// TwinCAT 3 PLC project Samples
// Title: TF8040 PLC-Samples
// Company: Beckhoff Automation GmbH
// Author: Beckhoff Automation
// ProjectVersion: 2.0.0.5
// Description: PLC.Samples to demontrate function volume of TF8040.
// ProgramVersion: 3.1.4023.0
// libraries:
//   Tc2_Standard, * (Beckhoff Automation GmbH)
//   Tc2_System, * (Beckhoff Automation GmbH)
//   Tc2_Utilities, * (Beckhoff Automation GmbH)
//   Tc3_BA2, * (Beckhoff Automation GmbH)
//   Tc3_BA2_Common, * (Beckhoff Automation GmbH)
//   Tc3_BACnetRev14, * (Beckhoff Automation GmbH)
//   Tc3_Module, * (Beckhoff Automation GmbH)
// project tree:
//   / PlcTask.TcTTO
//   SAMPLES/Demo/Event/ FB_Evt_Ack.TcPOU, FB_Evt_EventClasses.TcPOU, FB_Evt_Events.TcPOU, FB_Evt_Misc.TcPOU
//   SAMPLES/Demo/Objects/ FB_Obj_AddParam.TcPOU, FB_Obj_General.TcPOU, FB_Obj_Misc.TcPOU, FB_Obj_Sequence.TcPOU, FB_Obj_UserDefined.TcPOU
//   SAMPLES/Demo/Objects/Misc/ E_UDef_Mode.TcDUT (not stored), FB_UDef_BValEx.TcPOU (not stored), FB_UDef_SpVal.TcPOU (not stored), FB_UDef_SpValEx.TcPOU (not stored)
//   SAMPLES/Demo/Optional Extensions/Events/ FB_MyLocalObjectEvents.TcPOU
//   SAMPLES/Demo/Optional Extensions/ MAIN_OPTEXT.TcPOU
//   SAMPLES/Demo/Other/ FB_Misc.TcPOU
//   SAMPLES/Demo/Plant/ FB_Plt_Init1.TcPOU, FB_Plt_Init2.TcPOU, FB_Plt_Init3.TcPOU
//   SAMPLES/Demo/Reference/ FB_Ref_Collectors.TcPOU, FB_Ref_Groups.TcPOU
//   SAMPLES/Demo/Reference/Publish and Subscribe/ FB_Ref_PubSub_Local.TcPOU, FB_Ref_PubSub_Remote.TcPOU
//   SAMPLES/Demo/Structure/ FB_Struct_Nested.TcPOU
//   SAMPLES/Demo/Supplement specific/BACnet/ FB_BACnet_RcpList.TcPOU (not stored)
//   SAMPLES/Demo/[Helper]/FunctionBlocks/Aggregates/ FB_TimerAggregateA.TcPOU, FB_ProcAggregateB.TcPOU
//   SAMPLES/Demo/[Helper]/FunctionBlocks/Nested/ FB_NestedView.TcPOU, FB_NestedView2.TcPOU, FB_SubNestedView.TcPOU, FB_SubSubNestedView.TcPOU (not stored)
//   SAMPLES/ MAIN.TcPOU
//   SAMPLES/Templates/Standard/DUTs/Enumerations/OpMod/ E_OpMod_AC.TcDUT (not stored), E_OpMod_Binary.TcDUT, E_OpMod_ClsOpn.TcDUT (not stored), E_OpMod_Step2.TcDUT (not stored)
//   SAMPLES/Templates/Standard/GVLs/ MyLabels.TcGVL, MyProfiles.TcGVL
//   SAMPLES/Templates/Standard/POUs/Trade/General/Building/ FB_BA_Bld01.TcPOU (not stored)
//   SAMPLES/Templates/Standard/POUs/Trade/General/EventClasses/ FB_BA_EC01.TcPOU
//   SAMPLES/Templates/User-defined/Objects/ FB_UDef_Obj.TcPOU (not stored)
//   SAMPLES/Templates/User-defined/Sample Weather Station/ FB_BA_MyWeatherStation.TcPOU (not stored), FB_BA_MyWeatherStationSub.TcPOU (not stored), I_BA_MyWeatherStation.TcIO (not stored), ST_BA_MyWeatherData.TcDUT (not stored)
// real-time tasks:
//   TASK PlcTask: cycle T#45ms, priority 20, ADS port 350
//   TASK Device 1 (BACnet IP)_Task_58: cycle T#40ms, priority 58, ADS port 351
//   TASK Gerät 1 (BACnet IP)_QueueTask: cycle T#2ms, priority 8, ADS port 352
// I/O:
//   DEVICE Gerät 1 (BACnet IP), AmsNetId 192.168.216.1.2.1
// variable links:
//   Samples/Samples Instance <-> Device 1 (BACnet IP)
//     PlcTask Inputs/Tc3_BACnetRev14.BACnet_Globals.DefaultAdapter.BACnet_AmsNetId <-> Inputs/AmsNetId

CONFIGURATION Samples
    RESOURCE PLC ON TwinCAT3
        TASK PlcTask(INTERVAL := T#45ms, PRIORITY := 20);
        PROGRAM MAIN WITH PlcTask : MAIN;
    END_RESOURCE
END_CONFIGURATION

// ---- SAMPLES/Templates/Standard/DUTs/Enumerations/OpMod/E_OpMod_Binary.TcDUT
{attribute 'qualified_only'}
TYPE E_OpMod_Binary :
(
	eOff			:= 0,
	eOn				:= 1
	
) UDINT;
END_TYPE

// ---- SAMPLES/Templates/Standard/GVLs/MyLabels.TcGVL
{attribute 'qualified_only'}
VAR_GLOBAL
	{region 'Functions'}
		// A
		// B
		Cmd					: FB_BA_Label			:= (sObjName:='CMD',		sDescr:='Command');
		Col					: FB_BA_Label			:= (sObjName:='KUE',		sDescr:='Kühler');
		DmprEx				: FB_BA_Label			:= (sObjName:='KL',			sDescr:='Absperrklappe Abluft');
		DmprSu				: FB_BA_Label			:= (sObjName:='KL',			sDescr:='Absperrklappe Zuluft');
		Erc					: FB_BA_Label			:= (sObjName:='WRG',		sDescr:='Wärmerückgewinnung');
		EvtCl				: FB_BA_Label			:= (sObjName:='EC',			sDescr:='Eventklasse');
		FanEx				: FB_BA_Label			:= (sObjName:='VAB',		sDescr:='Abluftventilator');
		FanSu				: FB_BA_Label			:= (sObjName:='VZU',		sDescr:='Zuluftventilator');
		// G
		// H
		// I
		// J
		// K
		// L
		// M
		// N
		// O
		PltCtrl				: FB_BA_Label			:= (sObjName:='PC',			sDescr:='Anlagensteuerung');
		PreHtr				: FB_BA_Label			:= (sObjName:='LE',			sDescr:='Lufterhitzer');
		// Q
		// R
		// S	
		Trnd				: FB_BA_Label			:= (sObjName:='TR',			sDescr:='Trend');
		// U
		// v
		// W
		// X
		// Y
		// Z
	{endregion}
	{region 'Aggregates'}
		// A
		// B
		// C
		// D
		// E
		// F
		// G
		// H
		// I
		// J
		// K
		// L
		// M
		// N
		// O
		// P	
		// Q
		// R
		// S	
		// t
		// U
		// v
		// W
		// X
		// Y
		// Z
	{endregion}
	{region 'Processes'}
		ProcPreRinse		: FB_BA_LabelProcess	:= (sProcessName:='Vorspülen');
		ProcDriveDamper		: FB_BA_LabelProcess	:= (sProcessName:='Klappen fahren');
	{endregion}
END_VAR

// ---- SAMPLES/Templates/Standard/GVLs/MyProfiles.TcGVL
{attribute 'qualified_only'}
VAR_GLOBAL
	{region 'Placeholder'}
		{region 'Text'}
			txtOff						: STRING						:= 'Aus';
			txtOn						: STRING						:= 'Ein';
			txtNormal					: STRING						:= 'Normal';
			txtOffnormal				: STRING						:= 'Unnormal';
			txtAlert					: STRING						:= 'Alarm';
			txtDisturb					: STRING						:= 'Störung';
			txtExceeded					: STRING						:= 'Überschritten';
			txtMonitoring				: STRING						:= 'Überwachung';
			txtProtection				: STRING						:= 'Schutzbetrieb';
			txtEconomy					: STRING						:= 'Economy';
			txtComfort					: STRING						:= 'Comfort';
		{endregion}
		{region 'Event Transition Text'}
			trnsExceeded				: T_BA_EventTransitionText		:= [txtExceeded,			txtDisturb,			txtNormal];
			trnsMonitoring				: T_BA_EventTransitionText		:= [txtMonitoring,			txtDisturb,			txtNormal];
		{endregion}
		{region 'Multistate Text'}
			txtEnergyLevel				: T_BA_StateTextArray			:= [txtProtection,			txtEconomy,			txtComfort];
		{endregion}
	{endregion}
END_VAR
VAR_GLOBAL
	{region 'Sample Templates'}
		// A
		// B
		CmdB							: FB_BA_ProfileBEvtObj			:= (sInactiveText := txtOff,			sActiveText := txtOn,			aEventTransitionText := trnsMonitoring,							nEventClassID := 11);
		// D
		// E
		// F
		// G
		// H
		// I
		// J
		// K
		// L
		// M
		// N
		// O
		// P	
		// Q
		// R
		// S	
		// t
		// U
		// v
		// W
		// X
		// Y
		// Z
	{endregion}
	{region 'Sample Objects'}
		{region 'Analog'}
			AV_Prf						: FB_BA_ProfileAEvtObj			:= (eUnit:=E_BA_Unit.eTemperature_DegreesCelsius,						aEventTransitionText:=MyProfiles.trnsExceeded,					nEventClassID:=11);
			AVOp_Prf					: FB_BA_ProfileAObj				:= (eUnit:=E_BA_Unit.eTemperature_DegreesCelsius);
			AI_Prf						: FB_BA_ProfileAEvtObj			:= (eUnit:=E_BA_Unit.eTemperature_DegreesCelsius,						aEventTransitionText:=MyProfiles.trnsExceeded,					nEventClassID:=11);
			AO_Prf						: FB_BA_ProfileAEvtObj			:= (eUnit:=E_BA_Unit.eTemperature_DegreesCelsius,						aEventTransitionText:=MyProfiles.trnsExceeded,					nEventClassID:=11);
		{endregion}
		{region 'Binary'}
			BV_Prf						: FB_BA_ProfileBEvtObj			:= (sInactiveText := txtOff, sActiveText := txtOn,						aEventTransitionText:=MyProfiles.trnsExceeded,					nEventClassID:=11);
			BVOp_Prf					: FB_BA_ProfileBObj				:= (sInactiveText := txtOff, sActiveText := txtOn);
			BI_Prf						: FB_BA_ProfileBEvtObj			:= (sInactiveText := txtOff, sActiveText := txtOn,						aEventTransitionText:=MyProfiles.trnsExceeded,					nEventClassID:=11);
			BO_Prf						: FB_BA_ProfileBEvtObj			:= (sInactiveText := txtOff, sActiveText := txtOn,						aEventTransitionText:=MyProfiles.trnsExceeded,					nEventClassID:=11);
		{endregion}
		{region 'Multistate'}
			MV_Prf						: FB_BA_ProfileMEvtObj			:= (aStateText:=MyProfiles.txtEnergyLevel,								aEventTransitionText:=MyProfiles.trnsExceeded,					nEventClassID:=11);	
			MVOp_Prf					: FB_BA_ProfileMObj				:= (aStateText:=MyProfiles.txtEnergyLevel);
			MI_Prf						: FB_BA_ProfileMEvtObj			:= (aStateText:=MyProfiles.txtEnergyLevel,								aEventTransitionText:=MyProfiles.trnsExceeded,					nEventClassID:=11);
			MO_Prf						: FB_BA_ProfileMEvtObj			:= (aStateText:=MyProfiles.txtEnergyLevel,								aEventTransitionText:=MyProfiles.trnsExceeded,					nEventClassID:=11);
		{endregion}
		{region 'Misc'}
			Loop_Prf					: FB_BA_ProfileAObj				:= (eUnit:=E_BA_Unit.eOther_Percent);
			Cal_Prf						: FB_BA_ProfileBObj				:= (sInactiveText := txtOff, sActiveText := txtOn);
			SchedA_Prf					: FB_BA_ProfileAObj				:= (eUnit:=E_BA_Unit.eOther_Percent);
			SchedB_Prf					: FB_BA_ProfileBObj				:= (sInactiveText := txtOff, sActiveText := txtOn);
			SchedM_Prf					: FB_BA_ProfileMObj				:= (aStateText:=MyProfiles.txtEnergyLevel);
			Trend_Prf					: FB_BA_ProfileBObj				:= (sInactiveText := txtOff, sActiveText := txtOn);
			EvtCls_Prf					: FB_BA_Profile;
		{endregion}
		{region 'Custom'}
			MyWthSt_Prf					: FB_BA_Profile;
		{endregion}
		{region 'Collectors'}
			Col_PrfEn					: FB_BA_ProfileBObj				:= (sInactiveText := 'Nein', sActiveText := 'Ja');
			Col_PrfValA					: FB_BA_ProfileAObj				:= (eUnit:=E_BA_Unit.eTemperature_DegreesCelsius);
		{endregion}
	{endregion}
END_VAR

// ---- SAMPLES/MAIN.TcPOU
PROGRAM MAIN
VAR
	{region 'Settings'}
		DPAD					: FB_BA_CarelessDPAD:=(
									aIdentifier:=[
										(* Level 1 *)	(eNodeType:=E_BA_NodeType.eBuilding,	nIndexDigits:=2),
										(* Level 2 *)	(eNodeType:=E_BA_NodeType.eTrade,		nIndexDigits:=0),
										(* Level 3 *)	(eNodeType:=E_BA_NodeType.ePlant,		nIndexDigits:=2,			sSeparator_ObjectName:='~~~',		sSeparator_Description:=' --- '),
										(* Level 4 *)	(eNodeType:=E_BA_NodeType.eAggregate,	nIndexDigits:=2,			sSeparator_ObjectName:='++'),
										(* Level 5 *)	(eNodeType:=E_BA_NodeType.eFunction,	nIndexDigits:=3)
								]);
	{endregion}
		 
	Smpl						: FB_BA_View			:= (									sDescription:='Samples');
	{region 'Demonstration'}
		Demo					: FB_BA_View			:= (iParent:=Smpl,						sDescription:='Demonstration');
			Obj					: FB_BA_View			:= (iParent:=Demo,						sDescription:='Objects');
				General			: FB_Obj_General		:= (iParent:=Obj,						sDescription:='General objects');
				Misc			: FB_Obj_Misc			:= (iParent:=Obj,						sDescription:='Miscellaneous objects');
				Seq				: FB_Obj_Sequence		:= (iParent:=Obj,						sDescription:='Sequences');
				UdObj			: FB_Obj_UserDefined	:= (iParent:=Obj,						sDescription:='User defined objects');
				AddParam		: FB_Obj_AddParam		:= (iParent:=Obj,						sDescription:='Additional parameters');
					 
			Ref					: FB_BA_View			:= (iParent:=Demo,						sDescription:='Reference');
				Collect			: FB_Ref_Collectors		:= (iParent:=Ref,						sDescription:='Collectors');
				Groups			: FB_Ref_Groups			:= (iParent:=Ref,						sDescription:='Groups');
				PubSubLc		: FB_Ref_PubSub_Local	:= (iParent:=Ref,						sDescription:='Publisher and subscriber (Local)');
				PubSubRm		: FB_Ref_PubSub_Remote	:= (iParent:=Ref,						sDescription:='Publisher and subscriber (Remote)');
					 
			Evt					: FB_BA_View			:= (iParent:=Demo,						sDescription:='Event');
				EvtCls			: FB_Evt_EventClasses	:= (iParent:=Evt,						sDescription:='Event classes');
				Events			: FB_Evt_Events			:= (iParent:=Evt,						sDescription:='Events');
				Ack				: FB_Evt_Ack			:= (iParent:=Evt,						sDescription:='Acknowledgement');
				MiscEvt			: FB_Evt_Misc			:= (iParent:=Evt,						sDescription:='Miscellaneous');
					 
			Strct				: FB_BA_View			:= (iParent:=Demo,						sDescription:='Structure');
				Nested			: FB_Struct_Nested		:= (iParent:=Strct,						sDescription:='Nested objects');
					 
			Plt					: FB_BA_View			:= (iParent:=Demo,						sDescription:='Plant');
				PltCtrl1		: FB_Plt_Init1			:= (iParent:=Plt,						sDescription:='Plant control initialization 1');
				PltCtrl2		: FB_Plt_Init2			:= (iParent:=Plt,						sDescription:='Plant control initialization 2');
				PltCtrl3		: FB_Plt_Init3			:= (iParent:=Plt,						sDescription:='Plant control initialization 3');
					 
			Spl					: FB_BA_View			:= (iParent:=Demo,						sDescription:='Supplement specific');
				BACnet_RcpList	: FB_BACnet_RcpList		:= (iParent:=Spl,						sDescription:='Recipient list (BACnet)');
					 
			Other				: FB_BA_View			:= (iParent:=Demo,						sDescription:='Other');
				MscOth			: FB_Misc				:= (iParent:=Other,						sDescription:='Miscellaneous');
	{endregion}
	{region 'Templates'}
		Tmpl					: FB_BA_View			:= (iParent:=Smpl,						sDescription:='Templates');
			Gen					: FB_BA_View			:= (iParent:=Tmpl,						sDescription:='General');
				Bld01			: FB_BA_Bld01			:= (iParent:=Gen,						sDescription:='Building information');
				EvtCls01		: FB_BA_EC01			:= (iParent:=Gen,						sDescription:='Event Classes');
	{endregion}		
END_VAR
VAR		
	nCounter					: UDINT					:= 0;	
END_VAR

nCounter:=(nCounter+1);

Smpl();

// Demonstration:
Demo();

Obj();
General();
Misc();
Seq();
UdObj();
AddParam();

Ref();
Collect();
Groups();
PubSubLc();
PubSubRm();

Evt();
EvtCls();
Events();
Ack();
MiscEvt();

Strct();
Nested();

Plt();
PltCtrl1();
PltCtrl2();
PltCtrl3();

Spl();
BACnet_RcpList();

Other();
MscOth();

// Templates:
Tmpl();

Gen();
Bld01();
EvtCls01();

// Optional extensions:
MAIN_OPTEXT();

END_PROGRAM

// ---- SAMPLES/Demo/Objects/FB_Obj_General.TcPOU
// Demonstration of objects.
// > See "FB_BA_EC01" to view decleared event classes.
FUNCTION_BLOCK FB_Obj_General EXTENDS FB_BA_View
VAR
	{region 'Analog'}
		A										: FB_BA_View := (
													iParent									:= THIS^,
													sDescription							:= '{Analog objects}'
												);
			 
			// Intention:						Value
			AV									: FB_BA_AV := (
													iParent									:= A,
													sDescription							:= '{Analog Value}',
													eUnit									:= E_BA_Unit.eOther_Percent,
													nEventClassID							:= 11,
													stLowLimit								:= F_BA_Limit(TRUE, 0),
													stHighLimit								:= F_BA_Limit(TRUE, 50),
													stTimeDelay								:= F_BA_TimeDelay(1, 1),
													bEnPgm									:= TRUE,
													fValPgm									:= 10.0
												);
													
			// Intention:						Value for Display
			// Operation:						Display
			fAVDsp_ValuePgm						: REAL := 0;
			AVDsp								: FB_BA_AV_Op := (
													iParent									:= A,
													sObjectName								:= '{MyAvDsp}',
													sDescription							:= '{Sample AV Display}',
													eUnit									:= E_BA_Unit.eOther_Percent
												);	
			
			// Intention:						Value for Setpoint
			// Operation:						Setpoint
			AVSp								: FB_BA_AV_Op := (
													iParent									:= A,
													sDescription							:= '{Sample AV Setpoint}',
													eUnit									:= E_BA_Unit.eTemperature_DegreesCelsius,
													fValueRm								:= 3
												);
			bAVSp2_ValViaProp					: BOOL;
			fAVSp2_ValViaProp					: REAL;
			AVSp2								: FB_BA_AV_Op := (
													iParent									:= A,
													sDescription							:= '{Sample AV Setpoint 2}',
													eUnit									:= E_BA_Unit.eTemperature_DegreesCelsius,
													fValueRm								:= 3
												);
		
			// Intention:						Input
			// Hardware:						Process Data
			fAI_Proc_ValuePgm					: REAL := 20;
			AI_Proc								: FB_BA_AI := (
													iParent									:= A,
													sDescription							:= '{Sample AI (Process Data)}',
													sDeviceType								:= 'Analoger Eingang',
													eUnit									:= E_BA_Unit.eOther_Percent,
													nEventClassID							:= 11
												);
		
			// Intention:						Input
			// Hardware:						Raw Data
			AI_Raw								: FB_BA_AI_Raw := (
													iParent									:= A,
													sDescription							:= '{Sample AI (Raw)}',
													sDeviceType								:= 'Analoger Eingang',
													eUnit									:= E_BA_Unit.eOther_Percent,
													nEventClassID							:= 11
												);
		
			// Intention:						Input
			// Hardware:						I/O
			AI_IO								: FB_BA_AI_IO := (
													iParent									:= A,
													sDescription							:= '{Sample AI (IO)}',
													sDeviceType								:= 'Analoger Eingang',
													eUnit									:= E_BA_Unit.eOther_Percent,
													nEventClassID							:= 11
												);
												
			AI_IO_2_10V							: FB_BA_AI_IO := (
													iParent									:= A,
													sDescription							:= '{Sample AI (IO)}',
													sDeviceType								:= 'Analoger Eingang (2-10V)',
													eUnit									:= E_BA_Unit.eOther_Percent,
													nEventClassID							:= 11
												);
		
			// Intention:						Input
			// Hardware:						I/O
			AI_Temp								: FB_BA_AI_IOEx := (
													iParent									:= A,
													sDescription							:= '{Sample AI Temperaturfühler (Temp)}',
													sDeviceType								:= 'Temperaturfühler',
													eUnit									:= E_BA_Unit.eTemperature_DegreesCelsius,
													eSensor									:= E_BA_MeasuringElement.eNI1000,
													nEventClassID							:= 11
												);
		
			// Intention:						Input for Display
			// Operation:						Display
			// Hardware:						I/O
			// Parameter:						EventDetectionEnable = FALSE
			AIDsp_IO							: FB_BA_AI_IO := (
													iParent									:= A,
													sDescription							:= '{Sample AI Display (IO)}',
													sDeviceType								:= 'Analoger Eingang',
													eUnit									:= E_BA_Unit.eOther_Percent,
													bEventDetectionEnable					:= FALSE,
													nEventClassID							:= 11
												);
		
			// Intention:						Output
			// Hardware:						Process Data
			AO_CmdProc							: FB_BA_AO := (
													iParent									:= A,
													sDescription							:= '{Analog Befehl (Process Data)}',
													eUnit									:= E_BA_Unit.eOther_Percent,
													nEventClassID							:= 11
												);
		
			// Intention:						Output
			// Hardware:						Raw Data
			AO_CmdRaw							: FB_BA_AO_Raw := (
													iParent									:= A,
													sDescription							:= '{Analog Befehl (Raw Data)}',
													eUnit									:= E_BA_Unit.eOther_Percent,
													nEventClassID							:= 11
												);
		
			// Intention:						Output
			// Hardware:						I/O
			AO_CmdIO							: FB_BA_AO_IO := (
													iParent									:= A,
													sDescription							:= '{Analog Befehl (IO)}',
													eUnit									:= E_BA_Unit.eOther_Percent,
													nEventClassID							:= 11
												);
		
			// Intention:						Output for Display
			// Operation:						Display
			// Hardware:						I/O
			// Parameter:						EventDetectionEnable = FALSE
			AODisp_CmdIO						: FB_BA_AO_IO := (
													iParent									:= A,
													sDescription							:= '{Analog Befehl Display (IO)}',
													eUnit									:= E_BA_Unit.eOther_Percent,
													bEventDetectionEnable					:= FALSE,
													nEventClassID							:= 11
												);
	{endregion}
	{region 'Binary'}
		B										: FB_BA_View := (
													iParent									:= THIS^,
													sDescription							:= '{Binary objects}'
												);
			 
			// Intention:						Value
			BV									: FB_BA_BV := (
													iParent									:= B,
													sDescription							:= '{Binary Value}',
													sInactiveText							:= 'Aus',
													sActiveText								:= 'Ein',
													nEventClassID							:= 10
												);
															
			// Intention:						Value for Display
			// Operation:						Display
			bBVDsp_ValuePgm						: BOOL := FALSE;
			BVDsp								: FB_BA_BV_Op := (
													iParent									:= B,
													sDescription							:= '{Sample BV Display}',
													sInactiveText							:= 'Aus',
													sActiveText								:= 'Ein'
												);
			
			// Intention:						Value for Setpoint
			// Operation:						Setpoint
			BVSp								: FB_BA_BV_Op := (
													iParent									:= B,
													sDescription							:= '{Sample BV Setpoint}',
													sInactiveText							:= 'Aus',
													sActiveText								:= 'Ein',
													bValueRm								:= TRUE
												);
												
			// Intention:						Value for Setpoint
			// Operation:						Pushbutton
			nBVPushButton_Counter				: UINT;
			BVPushButton						: FB_BA_BV_Op := (
													iParent									:= B,
													sDescription							:= '{Sample BV Pushbutton}',
													sInactiveText							:= 'Aus',
													sActiveText								:= 'Ein',
													eToggleMode								:= E_BA_ToggleMode.ePushButton
												);
		
			// Intention:						Input
			// Hardware:						Process Data
			BI_Proc								: FB_BA_BI := (
													iParent									:= B,
													sDescription							:= '{Sample BI (Process Data)}',
													sDeviceType								:= 'Sicherung',
													sInactiveText							:= 'Normal',
													sActiveText								:= 'Ausgelöst',
													nEventClassID							:= 11
												);
		
			// Intention:						Input
			// Hardware:						Raw Data
			BI_Raw								: FB_BA_BI_Raw := (
													iParent									:= B,
													sDescription							:= '{Sample BI (Raw Data)}',
													sDeviceType								:= 'Sicherung',
													sInactiveText							:= 'Normal',
													sActiveText								:= 'Ausgelöst',
													nEventClassID							:= 11
												);
		
			// Intention:						Input
			// Hardware:						I/O
			BI_DstbIO							: FB_BA_BI_IO := (
													iParent									:= B,
													sDescription							:= '{Sample BI Disturb (IO)}',
													sDeviceType								:= 'Sicherung',
													sInactiveText							:= 'Normal',
													sActiveText								:= 'Ausgelöst',
													ePolarity								:= E_BA_Polarity.eReverse,
													nEventClassID							:= 51,
													eEnPlantLock							:= E_BA_LockPriority.eLocalMedium
												);
		
			// Intention:						Input for Display
			// Operation:						Display
			// Hardware:						I/O
			// Parameter:						EventDetectionEnable = FALSE
			BIDsp_SwiIO							: FB_BA_BI_IO := (
													iParent									:= B,
													sDescription							:= '{Sample BI Schalter Display (IO)}',
													sDeviceType								:= 'Sicherung',
													sInactiveText							:= 'Normal',
													sActiveText								:= 'Ausgelöst',
													ePolarity								:= E_BA_Polarity.eReverse,
													nEventClassID							:= 182,
													bEventDetectionEnable					:= FALSE
												);
		
			// Intention:						Output
			// Hardware:						I/O
			BO_CmdIO							: FB_BA_BO_IO := (
													iParent									:= B,
													sDescription							:= '{Sample BO Befehl (IO)}',
													sInactiveText							:= 'Aus',
													sActiveText								:= 'Ein',
													nEventClassID							:= 11,
													stTimeDelay := (
														nToAbnormal							:= 3
													)
												);
		
			// Intention:						Output
			// Hardware:						Process Data
			BO_CmdProc							: FB_BA_BO := (
													iParent									:= B,
													sDescription							:= '{Sample BO Befehl (Process Data)}',
													sInactiveText							:= 'Aus',
													sActiveText								:= 'Ein',
													nEventClassID							:= 11,
													stTimeDelay := (
														nToAbnormal							:= 3
													)
												);
		
			// Intention:						Output
			// Hardware:						Raw Data
			BO_CmdRaw							: FB_BA_BO_Raw := (
													iParent									:= B,
													sDescription							:= '{Sample BO Befehl (Raw Data)}',
													sInactiveText							:= 'Aus',
													sActiveText								:= 'Ein',
													nEventClassID							:= 11,
													stTimeDelay := (
														nToAbnormal							:= 3
													)
												);
													
			// Intention:						Output for Display
			// Operation:						Display
			// Hardware:						I/O
			// Parameter:						EventDetectionEnable = FALSE
			BODisp_CmdIO						: FB_BA_BO_IO := (
													iParent									:= B,
													sDescription							:= '{Sample BO Befehl Display (IO)}',
													sInactiveText							:= 'Aus',
													sActiveText								:= 'Ein',
													nEventClassID							:= 182,
													bEventDetectionEnable					:= FALSE
												);
	{endregion}
	{region 'Multistate'}
		M										: FB_BA_View := (
													iParent									:= THIS^,
													sDescription							:= '{Multistate objects}'
												);
			 
			// Intention:						Value
			MV									: FB_BA_MV := (
													iParent									:= M,
													sDescription							:= '{Sample MV}',
													aStateText								:= [ 'Aus', 'Stufe 1', 'Stufe 2' ],
													nEventClassID							:= 11
												);
			
			// Intention:						Value for Display
			// Operation:						Display
			nAVDsp_ValuePgm						: UDINT := 1;
			MVDsp								: FB_BA_MV_Op := (
													iParent									:= M,
													sObjectName								:= '{BAS01}',
													sDescription							:= '{Sample MV Display}',
													aStateText								:= [ 'Auto', 'Aus', 'Stufe 1', 'Stufe 2' ]
												);
			
			// Intention:						Value for Setpoint
			// Operation:						Setpoint
			MVSp								: FB_BA_MV_Op := (
													iParent									:= M,
													sObjectName								:= '{BAM01}',
													sDescription							:= '{Sample MV Setpoint}',
													aStateText								:= [ 'Auto', 'Aus', 'Stufe 1', 'Stufe 2' ],
													nValueRm								:= 1
												);
												
												
			nMVPushButton_Counter				: UDINT;
			MVPushButton						: FB_BA_MV_Op := (
													iParent									:= M,
													sDescription							:= '{Sample MV Pushbutton}',
													aStateText								:= [ 'Aus', 'Increment 1', 'Increment 2' ],
													eToggleMode								:= E_BA_ToggleMode.ePushButton
												);
		
			// Intention:						Input
			// Hardware:						Process Data
			MI_StateProc						: FB_BA_MI := (
													iParent									:= M,
													sDescription							:= '{Sample MI State (Process Data)}',
													sDeviceType								:= 'Gerät',
													aStateText								:= [ 'Aus', 'Stufe 1', 'Stufe 2', 'Stufe 3', 'Stufe 4' ],
													aAlarmValues							:= [ 3, 4 ],
													aFaultValues							:= [ 5 ],
													nEventClassID							:= 11
												);
		
			// Intention:						Input
			// Hardware:						Raw Data
			MI_StateRaw							: FB_BA_MI_Raw := (
													iParent									:= M,
													sDescription							:= '{Sample MI State (Raw Data)}',
													sDeviceType								:= 'Gerät',
													aStateText								:= [ 'Aus', 'Stufe 1', 'Stufe 2', 'Stufe 3', 'Stufe 4' ],
													aAlarmValues							:= [ 3, 4 ],
													aFaultValues							:= [ 5 ],
													nEventClassID							:= 11
												);
		
			// Intention:						Input
			// Hardware:						I/O
			MI_StateIO							: FB_BA_MI_IO := (
													iParent									:= M,
													sDescription							:= '{Sample MI State (IO)}',
													sDeviceType								:= 'Gerät',
													aStateText								:= [ 'Aus', 'Stufe 1', 'Stufe 2', 'Stufe 3', 'Stufe 4' ],
													aAlarmValues							:= [ 3, 4 ],
													aFaultValues							:= [ 5 ],
													nEventClassID							:= 11
												);
		
			// Intention:						Input for Display
			// Operation:						Display
			// Hardware:						I/O
			// Parameter:						EventDetectionEnable = FALSE
			MIDsp_Swi_StateIO					: FB_BA_MI_IO := (
													iParent									:= M,
													sDescription							:= '{Sample MI State (IO)}',
													sDeviceType								:= 'Gerät',
													aStateText								:= [ 'Zustand 1', 'Zustand 2', 'Zustand 3', 'Unbekannt' ],
													nEventClassID							:= 182,
													bEventDetectionEnable					:= FALSE
												);
		
			// Intention:						Output for Display
			// Operation:						Display
			// Hardware:						I/O
			// Parameter:						EventDetectionEnable = FALSE
			MODisp_IO							: FB_BA_MO_IO := (
													iParent									:= M,
													sDescription							:= '{Sample MO Befehl (IO)}',
													aStateText								:= [ 'Aus', 'Stufe 1', 'Stufe 2', 'Stufe 3', 'Stufe 4' ],
													nEventClassID							:= 182,
													bEventDetectionEnable					:= FALSE
												);
		
			// Intention:						Output
			// Hardware:						Process Data
			MO_CmdProc							: FB_BA_MO := (
													iParent									:= M,
													sDescription							:= '{Sample MO Befehl (Process Data)}',
													aStateText								:= [ 'Aus', 'Stufe 1', 'Stufe 2', 'Stufe 3', 'Stufe 4' ],
													nEventClassID							:= 182
												);
		
			// Intention:						Output
			// Hardware:						Raw Data
			MO_CmdRaw							: FB_BA_MO_Raw := (
													iParent									:= M,
													sDescription							:= '{Sample MO Befehl (Raw Data)}',
													aStateText								:= [ 'Aus', 'Stufe 1', 'Stufe 2', 'Stufe 3', 'Stufe 4' ],
													nEventClassID							:= 182
												);
	{endregion}
END_VAR

SUPER^();

// Analog:
A();

AV();
AVDsp(fValuePgm	:= MAX(fAVDsp_ValuePgm, AVSp.fPresentValue));
AVSp();
IF (bAVSp2_ValViaProp) THEN
	bAVSp2_ValViaProp := FALSE;
	AVSp2.PresentValue := fAVSp2_ValViaProp;
END_IF
AVSp2();
AI_Proc(fVal := fAI_Proc_ValuePgm);
AI_Raw();
AI_IO();
AI_IO_2_10V();
AI_Temp();
AIDsp_IO();
AO_CmdProc();
AO_CmdRaw();
AO_CmdIO();
AODisp_CmdIO();

// Binary:
B();

BV(bEnCrit := BI_DstbIO.bEvent);
BVDsp(bValuePgm	:= (bBVDsp_ValuePgm OR BVSp.bPresentValue));
BVSp();
BVPushButton();
BI_Proc();
BI_Raw();
BI_DstbIO();
BIDsp_SwiIO();
BO_CmdProc();
BO_CmdRaw();
BO_CmdIO();
BODisp_CmdIO();

IF (BVPushButton.bPresentValue <> BVPushButton.bDefaultValue) THEN
	nBVPushButton_Counter := (nBVPushButton_Counter+1);
END_IF

// Multistate:
M();

MV();
MVDsp(nValuePgm := MAX(nAVDsp_ValuePgm, MVSp.nPresentValue));
MVSp();
MVPushButton();
MI_StateProc();
MI_StateRaw();
MI_StateIO();
MIDsp_Swi_StateIO();
MODisp_IO(
	bEnPgm		:= TRUE,
	nValPgm		:= LIMIT(1, TO_UDINT(AVSp.fPresentValue), MODisp_IO.StateCount)
);
MO_CmdProc();
MO_CmdRaw();

IF (MVPushButton.nPresentValue <> MVPushButton.nDefaultValue) THEN
	nMVPushButton_Counter := (nMVPushButton_Counter+(MVPushButton.nPresentValue-1));
END_IF

END_FUNCTION_BLOCK

// ---- SAMPLES/Demo/Objects/FB_Obj_Misc.TcPOU
// Demonstration of objects.
// > See "FB_BA_EC01" to view decleared event classes.
FUNCTION_BLOCK FB_Obj_Misc EXTENDS FB_BA_View
VAR CONSTANT
	TREND_COUNT									: INT										:= 10;
END_VAR
VAR
	{region 'Project'}
		Proj									: FB_BA_View := (
													iParent									:= THIS^,
													sDescription							:= '{Project information}'
												);
				 
			// Intention:						Project Information
			Project								: FB_BA_Project := (
													iParent									:= Proj,
													sDescription							:= '{My project infos}',
													stProject := (	
														sTitle								:= 'Mein Projekt',
														sDescription						:= 'PLC Beispielprojekt',
														sLocation							:= 'Verl'
													)
												);
	{endregion}
	{region 'Loop'}
		Loop									: FB_BA_View := (
													iParent									:= THIS^,
													sDescription							:= '{Loop objects}'
												);
				 
			fLoop_Setpoint						: REAL										:= 20;								// Temperature setpoint.
			fLoop_CtrlVal						: REAL										:= 16;								// Simulation of controlled variable value.

			// Initialization:					Single loop for heating.
			Heat_En								: REFERENCE TO BOOL							REF= Heat.bEn;
			Heat_EnSync							: REFERENCE TO BOOL							REF= Heat.bEnSync;
			Heat_ValSync						: REFERENCE TO REAL							REF= Heat.fValSync;
			Heat_Y								: REFERENCE TO REAL							REF= Heat.fPresentValue;
			Heat								: FB_BA_Loop := (
													iParent									:= Loop,
													sDescription							:= '{Heating Loop}',
													eOutputUnit								:= E_BA_Unit.eOther_Percent,
													bEn										:= TRUE,
													eActionRm								:= E_BA_Action.eReverse,
													fProportionalConstant					:= 3.0,
													fIntegralConstant						:= 180
												);

			// Initialization:					Single loop for heating.
			Cool_En								: REFERENCE TO BOOL							REF= Cool.bEn;
			Cool_EnSync							: REFERENCE TO BOOL							REF= Cool.bEnSync;
			Cool_ValSync						: REFERENCE TO REAL							REF= Cool.fValSync;
			Cool_Y								: REFERENCE TO REAL							REF= Cool.fPresentValue;
			Cool								: FB_BA_Loop := (
													iParent									:= Loop,
													sDescription							:= '{Cooling Loop}',
													eOutputUnit								:= E_BA_Unit.eOther_Percent,
													bEn										:= TRUE,
													eActionRm								:= E_BA_Action.eDirect,
													fProportionalConstant					:= 3.0,
													fIntegralConstant						:= 180
												);
	{endregion}
	{region 'Calendar'}
		Cals									: FB_BA_View := (
													iParent									:= THIS^,
													sDescription							:= '{Calendar objects}'
												);

			// Intention:						Initialize calendar parameters with parameter builders.
			// Parameter:						tWeek										= F_BA_CalendarBuilder()
			Cal1								: FB_BA_Cal := (
													iParent									:= Cals,
													sDescription							:= '{Calendar 1}',
													aDateList								:= F_BA_CalendarBuilder()
																								.AppendDate(2021, E_BA_Month.eMarch, 10)
																								.AppendDateRange(nFromYear := 2021,E_BA_Month.eMarch,10, nToYear := 2021,E_BA_Month.eMarch,15)
																								.AppendWeekNDay(E_BA_Weekday.eMonday, E_BA_Week.Unspecified, E_BA_Month.Unspecified)
																								.Build()
												);
													 
			// Intention:						Initialize calendar parameters with helper methods.
			//									aDateList									= [(..., F_BA_DateVal(...)), (..., F_BA_DateRangeVal(...)), (..., F_BA_WeekNDayVal(...))]
			Cal2								: FB_BA_Cal := (
													iParent									:= Cals,
													sDescription							:= '{Calendar 2}',
													aDateList := [(
														eType								:= E_BA_DateValChoice.eDate,
														uDate								:= F_BA_DateVal(2020,E_BA_Month.eDecember,10)
													),(
														eType								:= E_BA_DateValChoice.eDateRange,
														uDate								:= F_BA_DateRangeVal(nFromYear:=2020,E_BA_Month.eMarch,5, nToYear:=2020,E_BA_Month.eMarch,10)
													),(
														eType								:= E_BA_DateValChoice.eWeekNDay,
														uDate								:= F_BA_WeekNDayVal(E_BA_Weekday.eTuesday, E_BA_Week.Unspecified, E_BA_Month.Unspecified)
													)]
												);

			Cal3								: FB_BA_Cal := (
													iParent									:= Cals,
													sDescription							:= '{Calendar 3}'
												);
	{endregion}
	{region 'Scheduler'}
		Sched									: FB_BA_View := (
													iParent									:= THIS^,
													sDescription							:= '{Schedule objects}'
												);
			
			// Intention:						Initialize scheduler parameters with parameter builders.
			// Parameter:						tWeek										= F_BA_WeeklyScheduleBuilder()
			//									tCalendar									= F_BA_ScheduleCalendarBuilder()
			//									tException									= F_BA_ExceptionScheduleBuilder()
			SchedA								: FB_BA_SchedA := (
													iParent									:= Sched,
													sDescription							:= '{Schedule Analog}',
													eUnit									:= E_BA_Unit.eTemperature_DegreesCelsius,
													aWeek									:= F_BA_WeeklyScheduleBuilder()
																								.SetAllDays()
																									.AppendA(T#0H, 1.0)
																									.Close()
																								.SetDay(E_BA_Weekday.eMonday)
																									.AppendA(T#0H, 2.0).AppendA(T#8H, 3.0).AppendA(T#16H, 2.0)
																									.Close()
																								.SetDayRange(E_BA_Weekday.eSaturday, E_BA_Weekday.eSunday)
																									.AppendA(T#0H, 4.0)
																									.Close()
																								.Build(),
													aCalendar								:= F_BA_ScheduleCalendarBuilder()
																								.AppendReference(Cal1)
																									.AppendA(T#0H, 1.0).AppendA(T#6H, 2.0).AppendNull(T#12H)
																									.Close()
																								.AppendReference(Cal2)
																									.AppendA(T#10H, 1.0).AppendNull(T#12H)
																									.Close()
																								.Build(),
													aException								:= F_BA_ExceptionScheduleBuilder()
																								.AppendDate(2021, E_BA_Month.eMarch, 10)
																									.AppendA(T#0H, 1.0).AppendA(T#6H, 2.0).AppendNull(T#12H)
																									.Close()
																								.AppendDateRange(nFromYear := 2021,E_BA_Month.eMarch,10, nToYear := 2021,E_BA_Month.eMarch,15)
																									.AppendA(T#12H, 1.0).AppendNull(T#16H)
																									.Close()
																								.AppendWeekNDay(E_BA_Weekday.eFriday, E_BA_Week.Unspecified, E_BA_Month.Unspecified)
																									.AppendA(T#20H, 3.0)
																									.Close()
																								.Build()
												);
			
			// Intention:						Initialize scheduler parameters with helper methods.
			// Parameter:						tWeek										= F_BA_SchedWeeklyXxA(...)
			//									tCalendar									= F_BA_SchedCalendar(...)
			//									tException									= [(..., F_BA_SchedEntryXxA(...)), (..., F_BA_SchedEntryXxA(...)), (..., F_BA_SchedEntryXxA(...))]
			SchedB								: FB_BA_SchedB := (
													iParent									:= Sched,
													sDescription							:= '{Schedule Bool}',
													sInactiveText							:= 'Aus',
													sActiveText								:= 'Ein',
													aWeek									:= F_BA_SchedWeekly3xB(E_BA_Weekday.eMonday, E_BA_Weekday.eFriday, T#0H, FALSE, T#6H, TRUE, T#20H, FALSE),
													aCalendar := [(
														iRefCalendar						:= Cal1,
														aEntry								:= F_BA_SchedEntry2xB(T#8H, TRUE, T#18H, FALSE)
													)],
													aException := [(
														eType								:= E_BA_DateValChoice.eDate,
														uDate								:= F_BA_DateVal(2021,E_BA_Month.eMarch,10),
														aEntry								:= F_BA_SchedEntry1xB(T#0H, FALSE)
													),(
														eType								:= E_BA_DateValChoice.eDateRange,
														uDate								:= F_BA_DateRangeVal(nFromYear:=2021,E_BA_Month.eMarch,10, nToYear:=2021,E_BA_Month.eMarch,15),
														aEntry								:= F_BA_SchedEntry2xB(T#10H, TRUE, T#17H, F_BA_NullB())
													),(
														eType								:= E_BA_DateValChoice.eWeekNDay,
														uDate								:= F_BA_WeekNDayVal(E_BA_Weekday.eFriday, E_BA_Week.Unspecified, E_BA_Month.Unspecified),
														aEntry								:= F_BA_SchedEntry3xB(T#9H, FALSE, T#12H, TRUE, T#17H, F_BA_NullB())
													)]);
			// Intention:						Initialize scheduler parameters manually.
			//									tCalendar									= ...
			//									tException									= ...
			SchedM								: FB_BA_SchedM := (
													iParent									:= Sched,
													sDescription							:= '{Schedule Multistate}',
													aStateText								:= [ 'Aus', 'Stufe 1', 'Stufe 2', 'Stufe 3' ],
													aWeek									:= F_BA_SchedWeekly3xM(E_BA_Weekday.eMonday, E_BA_Weekday.eFriday, T#0H, 1, T#6H, 2, T#20H, 1),
													aCalendar := [(
														iRefCalendar						:= Cal1,
														aEntry := [(
															eState							:= E_BA_SchedEntryState.eValue,
															stTime							:= F_BA_ToSTTime(T#16H),
															uValue							:= F_BA_UDIVal(2)
														),(
															eState							:= E_BA_SchedEntryState.eValue,
															stTime							:= F_BA_ToSTTime(T#20H),
															uValue							:= F_BA_UDIVal(1)
														)]
													)],
													aException := [(
														eType								:= E_BA_DateValChoice.eWeekNDay,
														uDate								:= F_BA_WeekNDayVal(E_BA_Weekday.eFriday, E_BA_Week.Unspecified, E_BA_Month.Unspecified),
														aEntry := [(
															eState							:= E_BA_SchedEntryState.eValue,
															stTime							:= F_BA_ToSTTime(T#10H),
															uValue							:= F_BA_UDIVal(2)
														),(
															eState							:= E_BA_SchedEntryState.eValue,
															stTime							:= F_BA_ToSTTime(T#12H),
															uValue							:= F_BA_UDIVal(3)
														),(
															eState							:= E_BA_SchedEntryState.eNull,
															stTime							:= F_BA_ToSTTime(T#16H)
														)]
													)]);
	{endregion}
	{region 'Trend'}
		Trnd									: FB_BA_View := (
													iParent									:= THIS^,
													sDescription							:= '{Trend objects}'
												);
				 
			// Intention:						Trend in polling-mode
			// Parameter:						eLoggingType								= E_BA_LoggingType.ePolled
			PollAV								: FB_BA_AV_Op := (
													iParent									:= Trnd,
													sDescription							:= '{Referenced object for polling}',
													eUnit									:= E_BA_Unit.eTemperature_DegreesCelsius,
													fValueRm								:= 3
												);
			TrendPoll							: FB_BA_Trend := (
													iParent									:= Trnd,
													sDescription							:= '{Sample Trend}',
													nEventClassID							:= 11,
													bEnable									:= TRUE,
													stStartTime								:= F_BA_ToSTDateTime(DT#2010-01-01-00:00),
													eLoggingType							:= E_BA_LoggingType.ePolled,
													nLogInterval							:= 300,
													stReferencedParam							:= F_BA_Reference(PollAV, E_BA_Parameter.ePresentValue)
												);
													
			// Intention:						Trend in trigger-mode
			// Parameter:						eLoggingType								= E_BA_LoggingType.ePolled
			TrigAV								: FB_BA_AV_Op := (
													iParent									:= Trnd,
													sDescription							:= '{Referenced object for polling}',
													eUnit									:= E_BA_Unit.eTemperature_DegreesCelsius,
													fValueRm								:= 1
												);
			TrendTrig_Man						: BOOL;
			TrendTrig							: FB_BA_Trend := (
													iParent									:= Trnd,
													sDescription							:= '{Sample Trend}',
													nEventClassID							:= 11,
													bEnable									:= TRUE,
													stStartTime								:= F_BA_ToSTDateTime(DT#2010-01-01-00:00),
													eLoggingType							:= E_BA_LoggingType.eTriggered,
													stReferencedParam						:= F_BA_Reference(TrigAV, E_BA_Parameter.ePresentValue)
												);
													 
			// Intention:						Trend in COV-mode
			// Parameter:						eLoggingType								= E_BA_LoggingType.eCOV
			CovAI								: FB_BA_AI := (
													iParent									:= Trnd,
													sDescription							:= '{Referenced analog object for COV}',
													eUnit									:= E_BA_Unit.eOther_Percent,
													nEventClassID							:= 11,
													bEventDetectionEnable					:= FALSE
												);
			TrendCovAI							: FB_BA_Trend := (
													iParent									:= Trnd,
													sDescription							:= '{Sample Analog Trend COV}',
													nEventClassID							:= 11,
													bEnable									:= TRUE,
													nBufferSize								:= 100,
													eLoggingType							:= E_BA_LoggingType.eCOV,
													stReferencedParam							:= F_BA_Reference(CovAI, E_BA_Parameter.ePresentValue)
												);
			CovBI								: FB_BA_BI := (
													iParent									:= Trnd,
													sDescription							:= '{Referenced binary object for COV}',
													sInactiveText							:= 'Off',
													sActiveText								:= 'On',
													nEventClassID							:= 11,
													bEventDetectionEnable					:= FALSE
												);
			TrendCovBI							: FB_BA_Trend := (
													iParent									:= Trnd,
													sDescription							:= '{Sample Binary Trend COV}',
													nEventClassID							:= 11,
													bEnable									:= TRUE,
													nBufferSize								:= 100,
													eLoggingType							:= E_BA_LoggingType.eCOV,
													stReferencedParam							:= F_BA_Reference(CovBI, E_BA_Parameter.ePresentValue)
												);
			CovMI								: FB_BA_MI := (
													iParent									:= Trnd,
													sDescription							:= '{Referenced multistate object for COV}',
													aStateText								:= ['Eco', 'Standard', 'Comfort'],
													nEventClassID							:= 11,
													bEventDetectionEnable					:= FALSE
												);
			TrendCovMI							: FB_BA_Trend := (
													iParent									:= Trnd,
													sDescription							:= '{Sample Multistate Trend COV}',
													nEventClassID							:= 11,
													bEnable									:= TRUE,
													nBufferSize								:= 100,
													eLoggingType							:= E_BA_LoggingType.eCOV,
													stReferencedParam							:= F_BA_Reference(CovMI, E_BA_Parameter.ePresentValue)
												);
													 
			// Intention:						Multiple trend objects as array
			Trends								: FB_BA_View := (
													iParent									:= Trnd,
													sDescription							:= 'Multiple trend objects'
												);
				Trend							: ARRAY[1 .. TREND_COUNT] OF FB_BA_Trend := [TREND_COUNT((
													iParent									:= Trends,
													iLabel									:= MyLabels.Trnd,
													nEventClassID							:= 11,
													eLoggingType							:= E_BA_LoggingType.eCOV
												))];
	{endregion}
END_VAR
VAR			
	_i											: INT;
END_VAR

SUPER^();

// Project:
Proj();

Project();

// Calendar:
Cals();

Cal1();
Cal2();
Cal3();

// Scheduler:
Sched();

SchedA();
SchedB();
SchedM();

// Loop:
Loop();

Heat(
	fSetpoint := fLoop_Setpoint,
	fCtrlVal := fLoop_CtrlVal
);
Cool(
	fSetpoint := fLoop_Setpoint,
	fCtrlVal := fLoop_CtrlVal
);

// Trend:
Trnd();

PollAV();
TrendPoll();
TrigAV(fValuePgm:=(TrigAV.fValuePgm+0.01));
TrendTrig(bTrigPgm:=((MAIN.nCounter MOD 250 = 0) OR (TrendTrig_Man)));
IF (MAIN.nCounter MOD 200 = 0) THEN
	CovAI.fVal := SEL((CovAI.fVal<10), 0, (CovAI.fVal+1));
END_IF
IF (MAIN.nCounter MOD 500 = 0) THEN
	CovBI.bVal := (NOT CovBI.bVal);
	CovMI.nVal := SEL((CovMI.nVal<CovMI.StateCount), 1, (CovMI.nVal+1));
END_IF
CovAI();
TrendCovAI();
CovBI();
TrendCovBI();
CovMI();
TrendCovMI();
Trends();
FOR _i := 1 TO TREND_COUNT DO
	Trend[_i]();
END_FOR

END_FUNCTION_BLOCK

// ---- SAMPLES/Demo/Objects/FB_Obj_Sequence.TcPOU
// Demonstration of objects.
// > See "FB_BA_EC01" to view decleared event classes.
FUNCTION_BLOCK FB_Obj_Sequence EXTENDS FB_BA_View
VAR
	{region 'Loop'}
		Loop									: FB_BA_View := (
													iParent									:= THIS^,
													sDescription							:= '{Loop objects}'
												);
				 
			// [Simulation]
			fLoop_Setpoint						: REAL										:= 20;								// Temperature setpoint.
			fLoop_Deadband						: REAL										:= 1.0;								// Deadband between heating- and cooling-loops.
			fLoop_CtrlVal						: REAL										:= 16;								// Simulation of controlled variable value.
			fLoop_ErcAction						: E_BA_Action								:= E_BA_Action.eDirect;				// Choose the ERC to be used for heating or cooling.
				 
			// [Sample 1.1]
			// Intention:						Mixed sequence of loops (heating an cooling)
			// Initialization:					Via sequence linker
			Seq1Heat2_En						: REFERENCE TO BOOL							REF= Seq1Heat2.bEn;
			Seq1Heat2_EnSync					: REFERENCE TO BOOL							REF= Seq1Heat2.bEnSync;
			Seq1Heat2_ValSync					: REFERENCE TO REAL							REF= Seq1Heat2.fValSync;
			Seq1Heat2_Y							: REFERENCE TO REAL							REF= Seq1Heat2.fPresentValue;
			Seq1Heat2							: FB_BA_LoopSeq := (
													iParent									:= Loop,
													sDescription							:= '{Heating Loop 2}',
													eOutputUnit								:= E_BA_Unit.eOther_Percent,
													bEn										:= TRUE,
													eActionRm								:= E_BA_Action.eReverse,
													fProportionalConstant					:= 3.0,
													fIntegralConstant						:= 180
												);
			Seq1Heat1_En						: REFERENCE TO BOOL							REF= Seq1Heat1.bEn;
			Seq1Heat1_EnSync					: REFERENCE TO BOOL							REF= Seq1Heat1.bEnSync;
			Seq1Heat1_ValSync					: REFERENCE TO REAL							REF= Seq1Heat1.fValSync;
			Seq1Heat1_Y							: REFERENCE TO REAL							REF= Seq1Heat1.fPresentValue;
			Seq1Heat1							: FB_BA_LoopSeq := (
													iParent									:= Loop,
													sDescription							:= '{Heating Loop 1}',
													eOutputUnit								:= E_BA_Unit.eOther_Percent,
													bEn										:= TRUE,
													eActionRm								:= E_BA_Action.eReverse,
													fProportionalConstant					:= 4.0,
													fIntegralConstant						:= 120
												);
			Seq1Erc_En							: REFERENCE TO BOOL							REF= Seq1Erc.bEn;
			Seq1Erc_EnSync						: REFERENCE TO BOOL							REF= Seq1Erc.bEnSync;
			Seq1Erc_ValSync						: REFERENCE TO REAL							REF= Seq1Erc.fValSync;
			Seq1Erc_Y							: REFERENCE TO REAL							REF= Seq1Erc.fPresentValue;
			Seq1Erc								: FB_BA_LoopSeq := (
													iParent									:= Loop,
													sDescription							:= '{ERC Loop 1}',
													eOutputUnit								:= E_BA_Unit.eOther_Percent,
													bEn										:= TRUE,
													eActionRm								:= E_BA_Action.eReverse,
													fProportionalConstant					:= 5.0,
													fIntegralConstant						:= 60
												);
			Seq1Cool_En							: REFERENCE TO BOOL							REF= Seq1Cool.bEn;
			Seq1Cool_EnSync						: REFERENCE TO BOOL							REF= Seq1Cool.bEnSync;
			Seq1Cool_ValSync					: REFERENCE TO REAL							REF= Seq1Cool.fValSync;
			Seq1Cool_Y							: REFERENCE TO REAL							REF= Seq1Cool.fPresentValue;
			Seq1Cool							: FB_BA_LoopSeq := (
													iParent									:= Loop,
													sDescription							:= '{Cooling Loop}',
													eOutputUnit								:= E_BA_Unit.eOther_Percent,
													bEn										:= TRUE,
													eActionRm								:= E_BA_Action.eDirect,
													fProportionalConstant					:= 4.0,
													fIntegralConstant						:= 60
												);
			Seq1_En								: REFERENCE TO BOOL							REF= Seq1.bEn;
			Seq1_Step							: REFERENCE TO STRING						REF= Seq1.sStep;
			Seq1								: FB_BA_SequenceLink := (
													iParent									:= Loop,
													sDescription							:= '{Mixed sequence}',
													iReference								:= [ Seq1Heat2, Seq1Heat1, Seq1Erc, Seq1Cool ]
												);
						
			// [Sample 1.2]							
			// Initialization:					Manual (No sequence linker used)
			// Parameter:						iNextSequenceRef = [reference to next loop]
			(*
			Seq1Heat2							: FB_BA_LoopSeq								:= (iNextSequenceRef := Seq1Heat1);
			Seq1Heat1							: FB_BA_LoopSeq								:= (iNextSequenceRef := Seq1Erc);
			Seq1Erc								: FB_BA_LoopSeq								:= (iNextSequenceRef := Seq1Cool);
			Seq1Cool							: FB_BA_LoopSeq;
			*) 

			// [Sample 2.1]
			// Intention:						Sequence of equal loops (heating)
			// Initialization:					Via sequence linker
			Seq2Heat3_En						: REFERENCE TO BOOL							REF= Seq2Heat3.bEn;
			Seq2Heat3_EnSync					: REFERENCE TO BOOL							REF= Seq2Heat3.bEnSync;
			Seq2Heat3_ValSync					: REFERENCE TO REAL							REF= Seq2Heat3.fValSync;
			Seq2Heat3_Y							: REFERENCE TO REAL							REF= Seq2Heat3.fPresentValue;
			Seq2Heat3							: FB_BA_LoopSeq := (
													iParent									:= Loop,
													sDescription							:= '{Heating Loop 3}',
													eOutputUnit								:= E_BA_Unit.eOther_Percent,
													bEn										:= TRUE,
													eActionRm								:= E_BA_Action.eReverse,
													fProportionalConstant					:= 1.0,
													fIntegralConstant						:= 180
												);
			Seq2Heat2_En						: REFERENCE TO BOOL							REF= Seq2Heat2.bEn;
			Seq2Heat2_EnSync					: REFERENCE TO BOOL							REF= Seq2Heat2.bEnSync;
			Seq2Heat2_ValSync					: REFERENCE TO REAL							REF= Seq2Heat2.fValSync;
			Seq2Heat2_Y							: REFERENCE TO REAL							REF= Seq2Heat2.fPresentValue;
			Seq2Heat2							: FB_BA_LoopSeq := (
													iParent									:= Loop,
													sDescription							:= '{Heating Loop 2}',
													eOutputUnit								:= E_BA_Unit.eOther_Percent,
													bEn										:= TRUE,
													eActionRm								:= E_BA_Action.eReverse,
													fProportionalConstant					:= 2.0,
													fIntegralConstant						:= 120
												);
			Seq2Heat1_En						: REFERENCE TO BOOL							REF= Seq2Heat1.bEn;
			Seq2Heat1_EnSync					: REFERENCE TO BOOL							REF= Seq2Heat1.bEnSync;
			Seq2Heat1_ValSync					: REFERENCE TO REAL							REF= Seq2Heat1.fValSync;
			Seq2Heat1_Y							: REFERENCE TO REAL							REF= Seq2Heat1.fPresentValue;
			Seq2Heat1							: FB_BA_LoopSeq := (
													iParent									:= Loop,
													sDescription							:= '{Heating Loop 1}',
													eOutputUnit								:= E_BA_Unit.eOther_Percent,
													bEn										:= TRUE,
													eActionRm								:= E_BA_Action.eReverse,
													fProportionalConstant					:= 3.0,
													fIntegralConstant						:= 60
												);
			Seq2_En								: REFERENCE TO BOOL							REF= Seq2.bEn;
			Seq2_Step							: REFERENCE TO STRING						REF= Seq2.sStep;
			Seq2								: FB_BA_SequenceLink := (
													iParent									:= Loop,
													sDescription							:= '{Heating sequence}',
													iReference								:= [ Seq2Heat3, Seq2Heat2, Seq2Heat1 ]
												);
						
			// [Sample 2.2]							
			// Initialization:					Manual (No sequence linker used)
			// Parameter:						iNextSequenceRef = [reference to next loop]
			(*
			Seq2Heat3							: FB_BA_LoopSeq								:= (iNextSequenceRef := Seq2Heat2);
			Seq2Heat2							: FB_BA_LoopSeq								:= (iNextSequenceRef := Seq2Heat1);
			Seq2Heat1							: FB_BA_LoopSeq;
			*)
				 
			// [Sample 3.1]
			// Intention:						Sequence of equal loops (Cooling)
			// Initialization:					Via sequence linker
			Seq3Cool1_En						: REFERENCE TO BOOL							REF= Seq3Cool1.bEn;
			Seq3Cool1_EnSync					: REFERENCE TO BOOL							REF= Seq3Cool1.bEnSync;
			Seq3Cool1_ValSync					: REFERENCE TO REAL							REF= Seq3Cool1.fValSync;
			Seq3Cool1_Y							: REFERENCE TO REAL							REF= Seq3Cool1.fPresentValue;
			Seq3Cool1							: FB_BA_LoopSeq := (
													iParent									:= Loop,
													sDescription							:= '{Cooling Loop 1}',
													eOutputUnit								:= E_BA_Unit.eOther_Percent,
													bEn										:= TRUE,
													eActionRm								:= E_BA_Action.eDirect,
													fProportionalConstant					:= 3.0,
													fIntegralConstant						:= 60
												);
			Seq3Cool2_En						: REFERENCE TO BOOL							REF= Seq3Cool2.bEn;
			Seq3Cool2_EnSync					: REFERENCE TO BOOL							REF= Seq3Cool2.bEnSync;
			Seq3Cool2_ValSync					: REFERENCE TO REAL							REF= Seq3Cool2.fValSync;
			Seq3Cool2_Y							: REFERENCE TO REAL							REF= Seq3Cool2.fPresentValue;
			Seq3Cool2							: FB_BA_LoopSeq := (
													iParent									:= Loop,
													sDescription							:= '{Cooling Loop 2}',
													eOutputUnit								:= E_BA_Unit.eOther_Percent,
													bEn										:= TRUE,
													eActionRm								:= E_BA_Action.eDirect,
													fProportionalConstant					:= 2.0,
													fIntegralConstant						:= 120
												);
			Seq3Cool3_En						: REFERENCE TO BOOL							REF= Seq3Cool3.bEn;
			Seq3Cool3_EnSync					: REFERENCE TO BOOL							REF= Seq3Cool3.bEnSync;
			Seq3Cool3_ValSync					: REFERENCE TO REAL							REF= Seq3Cool3.fValSync;
			Seq3Cool3_Y							: REFERENCE TO REAL							REF= Seq3Cool3.fPresentValue;
			Seq3Cool3							: FB_BA_LoopSeq := (
													iParent									:= Loop,
													sDescription							:= '{Cooling Loop 3}',
													eOutputUnit								:= E_BA_Unit.eOther_Percent,
													bEn										:= TRUE,
													eActionRm								:= E_BA_Action.eDirect,
													fProportionalConstant					:= 1.0,
													fIntegralConstant						:= 180
												);
			Seq3_En								: REFERENCE TO BOOL							REF= Seq3.bEn;
			Seq3_Step							: REFERENCE TO STRING						REF= Seq3.sStep;
			Seq3								: FB_BA_SequenceLink := (
													iParent									:= Loop,
													sDescription							:= '{Cooling sequence}',
													iReference								:= [ Seq3Cool1, Seq3Cool2, Seq3Cool3 ]
												);
						
			// [Sample 3.2]							
			// Initialization:					Manual (No sequence linker used)
			// Parameter:						iNextSequenceRef = [reference to next loop]
			(*
			Seq3Cool1							: FB_BA_LoopSeq								:= (iNextSequenceRef := Seq3Cool2);
			Seq3Cool2							: FB_BA_LoopSeq								:= (iNextSequenceRef := Seq3Cool3);
			Seq3Cool3							: FB_BA_LoopSeq;
			*)
	{endregion}
END_VAR
VAR
	_fSpH										: REAL;
	_fSpC										: REAL;
	_fSpErc										: REAL;
END_VAR

SUPER^();

Loop();

_fSpH := (fLoop_Setpoint - (fLoop_Deadband / 2));
_fSpC := (fLoop_Setpoint + (fLoop_Deadband / 2));
_fSpErc := SEL((fLoop_ErcAction = E_BA_Action.eDirect), _fSpH, _fSpC);

// [Sample 1.1]
Seq1Heat2(
	fSetpoint := _fSpH,
	fCtrlVal := fLoop_CtrlVal
);
Seq1Heat1(
	fSetpoint := _fSpH,
	fCtrlVal := fLoop_CtrlVal
);
Seq1Erc(
	fSetpoint := _fSpErc,
	fCtrlVal := fLoop_CtrlVal,
	eActionRm := fLoop_ErcAction
);
Seq1Cool(
	fSetpoint := _fSpC,
	fCtrlVal := fLoop_CtrlVal
);
Seq1();

// [Sample 2.1]
Seq2Heat3(
	fSetpoint := _fSpH,
	fCtrlVal := fLoop_CtrlVal
);
Seq2Heat2(
	fSetpoint := _fSpH,
	fCtrlVal := fLoop_CtrlVal
);
Seq2Heat1(
	fSetpoint := _fSpH,
	fCtrlVal := fLoop_CtrlVal
);
Seq2();

// [Sample 3.1]
Seq3Cool3(
	fSetpoint := _fSpH,
	fCtrlVal := fLoop_CtrlVal
);
Seq3Cool2(
	fSetpoint := _fSpH,
	fCtrlVal := fLoop_CtrlVal
);
Seq3Cool1(
	fSetpoint := _fSpH,
	fCtrlVal := fLoop_CtrlVal
);
Seq3();

END_FUNCTION_BLOCK

// ---- SAMPLES/Demo/Objects/FB_Obj_UserDefined.TcPOU
// Demonstration of objects.
// > See "FB_BA_EC01" to view decleared event classes.
FUNCTION_BLOCK FB_Obj_UserDefined EXTENDS FB_BA_View
VAR
	Misc					: FB_BA_View := (
								iParent					:= THIS^,
								sDescription			:= '{Miscellaneous use cases}'
							);
										
		// Intention:		Some object with some individual PLC logic (Will be is visible to clients like TcHmiBa, etc.)
		Obj1				: FB_UDef_Obj := (
								iParent					:= Misc,
								sDescription			:= '{Simple user defined object}'
							);
END_VAR

SUPER^();

Misc();

Obj1();

END_FUNCTION_BLOCK

// ---- SAMPLES/Demo/Objects/FB_Obj_AddParam.TcPOU
FUNCTION_BLOCK FB_Obj_AddParam EXTENDS FB_BA_View
VAR
	TestAVal			: FB_UDef_AVal				:= (iParent:=THIS^,		sDescription:='My user defined analog object',				eMode:=E_UDef_Mode.eAdd);
	TestAValEx			: FB_UDef_AValEx			:= (iParent:=THIS^,		sDescription:='Another user defined enabled analog object',	eMode:=E_UDef_Mode.eSubstract);
END_VAR
VAR
	{region 'Test'}
		nOffset			: UINT						:= 3;
	{endregion}
END_VAR

SUPER^(); // FB_BA_View
TestAVal(nSomeOffset := nOffset); // FB_UDef_AVal
TestAValEx(nSomeOffset := nOffset); // FB_UDef_AValEx

END_FUNCTION_BLOCK

// ---- SAMPLES/Demo/Reference/FB_Ref_Collectors.TcPOU
// Examples of collectors.
// [Hint]
// > All reference-variables are implemented to ease monitoring of relevant variables.
FUNCTION_BLOCK FB_Ref_Collectors EXTENDS FB_BA_View
VAR
	{region 'Analog'}
		_ValueA1					: REFERENCE TO REAL				REF= ValueA1.fValueRm;
		ValueA1						: FB_BA_AV_Op := (
										iParent						:= THIS^,
										iProfile					:= MyProfiles.AVOp_Prf,
										fValueRm					:= 0.0
									);
		_ValueA2					: REFERENCE TO REAL				REF= ValueA2.fValueRm;
		ValueA2						: FB_BA_AV_Op := (
										iParent						:= THIS^,
										iProfile					:= MyProfiles.AVOp_Prf,
										fValueRm					:= 1.0
									);
		ColectA						: FB_BA_Collector				:= (iParent:=THIS^, iReferences:=[ ValueA1, ValueA2 ]);
	{endregion}
	{region 'Binary'}
		_ValueB1					: REFERENCE TO BOOL				REF= ValueB1.bValueRm;
		ValueB1						: FB_BA_BV_Op := (
										iParent						:= THIS^,
										iProfile					:= MyProfiles.BVOp_Prf,
										bValueRm					:= FALSE
									);
		_ValueB2					: REFERENCE TO BOOL				REF= ValueB2.bValueRm;
		ValueB2						: FB_BA_BV_Op := (
										iParent						:= THIS^,
										iProfile					:= MyProfiles.BVOp_Prf,
										bValueRm					:= TRUE
									);
		ColectB						: FB_BA_Collector				:= (iParent:=THIS^, iReferences:=[ ValueB1, ValueB2 ]);
	{endregion}
	{region 'Multistate'}
		_ValueM1					: REFERENCE TO UDINT			REF= ValueM1.nValueRm;
		ValueM1						: FB_BA_MV_Op := (
										iParent						:= THIS^,
										iProfile					:= MyProfiles.MVOp_Prf,
										nValueRm					:= 1
									);
		_ValueM2					: REFERENCE TO UDINT			REF= ValueM2.nValueRm;
		ValueM2						: FB_BA_MV_Op := (
										iParent						:= THIS^,
										iProfile					:= MyProfiles.MVOp_Prf,
										nValueRm					:= 2
									);
		ColectM						: FB_BA_Collector				:= (iParent:=THIS^, iReferences:=[ ValueM1, ValueM2 ]);
	{endregion}
	{region 'View'}
		View1						: FB_BA_View					:= (iParent:=THIS^, sObjectName:='View1');
			_Enable1				: REFERENCE TO BOOL				REF= Enable1.bValueRm;	
			Enable1					: FB_BA_BV_Op := (
										iParent						:= View1,
										iProfile					:= MyProfiles.BVOp_Prf,
										bValueRm					:= FALSE
									);
			_Value1					: REFERENCE TO REAL				REF= Value1.fValueRm;
			Value1					: FB_BA_AV_Op := (
										iParent						:= View1,
										iProfile					:= MyProfiles.AVOp_Prf,
										fValueRm					:= 0.0
									);
		View2						: FB_BA_View					:= (iParent:=THIS^, sObjectName:='View2');
			_Enable01				: REFERENCE TO BOOL				REF= Enable01.bValueRm;	
			Enable01				: FB_BA_BV_Op := (
										iParent						:= View2,
										iProfile					:= MyProfiles.BVOp_Prf,
										bValueRm					:= TRUE
									);
			_Value01				: REFERENCE TO REAL				REF= Value01.fValueRm;
			Value01					: FB_BA_AV_Op := (
										iParent						:= View2,
										iProfile					:= MyProfiles.AVOp_Prf,
										fValueRm					:= 3.0
									);
		View3						: FB_NestedView					:= (View:=(iParent:=THIS^, sObjectName:='View3'));
			_Enable3				: REFERENCE TO BOOL				REF= View3.Enable.bValueRm;
			_Value3					: REFERENCE TO REAL				REF= View3.Value.fValueRm;
		View4						: FB_SubNestedView				:= (iParent:=THIS^, sObjectName:='View4');
			_Enable4				: REFERENCE TO BOOL				REF= View4.SubView.Enable.bValueRm;
			_Value4					: REFERENCE TO REAL				REF= View4.SubView.Value.fValueRm;
					  
		ColectEnA					: FB_BA_Collector := (
										iParent						:= THIS^,
										iReferences					:= [ View1, View2, View3.View ],
					  					sRefSubjectEn				:= 'Enable',							// <- Specified subject.
					  					sRefSubjectVal				:= 'Value'								// <- Specified subject.
									);
		ColectEnB					: FB_BA_Collector := (
										iParent						:= THIS^,
										iReferences					:= [ View4 ],
					  					sRefSubjectEn				:= 'SubView.Enable',					// <- Specified subject path.
					  					sRefSubjectVal				:= 'SubView.Value'						// <- Specified subject path.
									);
	{endregion}
END_VAR

SUPER^(); // FB_BA_View
ValueA1(); // FB_BA_AV_Op
ValueA2(); // FB_BA_AV_Op
ValueB1(); // FB_BA_BV_Op
ValueB2(); // FB_BA_BV_Op
ValueM1(); // FB_BA_MV_Op
ValueM2(); // FB_BA_MV_Op
View1(); // FB_BA_View
Enable1(); // FB_BA_BV_Op
Value1(); // FB_BA_AV_Op
View2(); // FB_BA_View
Enable01(); // FB_BA_BV_Op
Value01(); // FB_BA_AV_Op
View3(); // FB_NestedView
View4(); // FB_SubNestedView
ColectA(); // FB_BA_Collector
ColectB(); // FB_BA_Collector
ColectM(); // FB_BA_Collector
ColectEnA(); // FB_BA_Collector
ColectEnB(); // FB_BA_Collector

END_FUNCTION_BLOCK

// ---- SAMPLES/Demo/[Helper]/FunctionBlocks/Nested/FB_NestedView.TcPOU
FUNCTION_BLOCK FB_NestedView
VAR_INPUT CONSTANT
	View		: FB_BA_View;
		Enable	: FB_BA_BV_Op := (
					iParent			:= View,
					iProfile		:= MyProfiles.BVOp_Prf,
					bValueRm		:= FALSE
				);		
		Value	: FB_BA_AV_Op := (
					iParent			:= View,
					iProfile		:= MyProfiles.AVOp_Prf,
					fValueRm		:= 0.0
				);	
END_VAR

View();
Enable();
Value();

END_FUNCTION_BLOCK

// ---- SAMPLES/Demo/[Helper]/FunctionBlocks/Nested/FB_SubNestedView.TcPOU
FUNCTION_BLOCK FB_SubNestedView EXTENDS FB_BA_View
VAR_INPUT CONSTANT
	SubView		: FB_NestedView		:= (View := (iParent:=THIS^));
END_VAR

SUPER^();

SubView();

END_FUNCTION_BLOCK

// ---- SAMPLES/Demo/Reference/FB_Ref_Groups.TcPOU
// Examples of groups.
FUNCTION_BLOCK FB_Ref_Groups EXTENDS FB_BA_View
VAR
	{region 'Analog'}
		A							: FB_BA_View := (
										iParent							:= THIS^,
										sDescription					:= '{Analog objects}'
									);
				                    
			GrpAV1					: FB_BA_AV := (
										iParent							:= A,
										eUnit							:= E_BA_Unit.eOther_NoUnits,
										nEventClassID					:= 11,
										bEnPgm							:= TRUE,
										fValPgm							:= 10
									);
			GrpAV2					: FB_BA_AV := (
										iParent							:= A,
										eUnit							:= E_BA_Unit.eOther_NoUnits,
										nEventClassID					:= 11,
										bEnPgm							:= TRUE,
										fValPgm							:= 15
									);
			GrpAVOp1				: FB_BA_AV_Op := (
										iParent							:= A,
										eUnit							:= E_BA_Unit.eTemperature_DegreesCelsius,
										fValueRm						:= 20
									);
			GrpAVOp2				: FB_BA_AV_Op := (
										iParent							:= A,
										eUnit							:= E_BA_Unit.eTemperature_DegreesCelsius,
										fValueRm						:= 25
									);
										 
			// Intention:			Eigenständige Gruppe (Ohne Achsen-Zugehörigkeit)
			Group_AVMin				: FB_BA_Group_AVal := (
										eCalcMode						:= E_BA_AValCalcMode.eMin,
										iReference						:= [ GrpAV1, GrpAV2, GrpAVOp1, GrpAVOp2 ]
									);
			Group_AVMax				: FB_BA_Group_AVal := (
										eCalcMode						:= E_BA_AValCalcMode.eMax,
										iReference						:= [ GrpAV1, GrpAV2, GrpAVOp1, GrpAVOp2 ]
									);
			Group_AVAvg				: FB_BA_Group_AVal := (
										eCalcMode						:= E_BA_AValCalcMode.eAverage,
										iReference						:= [ GrpAV1, GrpAV2, GrpAVOp1, GrpAVOp2 ]
									);
	{endregion}
END_VAR

SUPER^(); // FB_BA_View
A(); // FB_BA_View
GrpAV1(); // FB_BA_AV
GrpAV2(); // FB_BA_AV
GrpAVOp1(); // FB_BA_AV_Op
GrpAVOp2(); // FB_BA_AV_Op
Group_AVMin(); // FB_BA_Group_AVal
Group_AVMax(); // FB_BA_Group_AVal
Group_AVAvg(); // FB_BA_Group_AVal

END_FUNCTION_BLOCK

// ---- SAMPLES/Demo/Reference/Publish and Subscribe/FB_Ref_PubSub_Local.TcPOU
// Example of internal device communication.
FUNCTION_BLOCK FB_Ref_PubSub_Local EXTENDS FB_BA_View
VAR
	{region 'Analog'}
	
		A								: FB_BA_View := (
											iParent						:= THIS^,
											sDescription				:= '{Analog objects}'
										);
													 
			AV_Sub						: FB_BA_SubAPrio				:= (sSubject:='AV_Obj');
			AV_Obj						: FB_BA_AV := (
											iParent						:= A,
											iProfile					:= MyProfiles.AV_Prf,
											bEnPublish					:= TRUE
										); 
			AVOp_Sub					: FB_BA_SubAV_Op				:= (sSubject:='AVOp_Obj');
			AVOp_Obj					: FB_BA_AV_Op := (
											iParent						:= A,
											iProfile					:= MyProfiles.AVOp_Prf,
											bEnPublish					:= TRUE,
											fValueRm					:= 10
										); 
			AI_Sub						: FB_BA_SubAI					:= (sSubject:='AI_Obj');
			AI_Obj						: FB_BA_AI_Raw := (
											iParent						:= A,
											iProfile					:= MyProfiles.AI_Prf,
											bEnPublish					:= TRUE
										); 
			AO_Sub						: FB_BA_SubAPrio				:= (sSubject:='AO_Obj');
			AO_Obj						: FB_BA_AO_Raw := (
											iParent						:= A,
											iProfile					:= MyProfiles.AO_Prf,
											bEnPublish					:= TRUE
										); 
	{endregion}
	{region 'Binary'}
		B								: FB_BA_View := (
											iParent						:= THIS^,
											sDescription				:= '{Binary objects}'
										);
												 
			BV_Sub						: FB_BA_SubBPrio				:= (sSubject:='BV_Obj'); 
			BV_Obj						: FB_BA_BV := (
											iParent						:= B,
											iProfile					:= MyProfiles.BV_Prf,
											bEnPublish					:= TRUE
										);
			BVOp_Sub					: FB_BA_SubBV_Op				:= (sSubject:='BVOp_Obj');
			BVOp_Obj					: FB_BA_BV_Op := (
											iParent						:= B,
											iProfile					:= MyProfiles.BVOp_Prf,
											bEnPublish					:= TRUE,
											bValueRm					:= TRUE
										);
			BI_Sub						: FB_BA_SubBI					:= (sSubject:='BI_Obj');
			BI_Obj						: FB_BA_BI_Raw := (
											iParent						:= B,
											iProfile					:= MyProfiles.BI_Prf,
											bEnPublish					:= TRUE
										);
			BO_Sub						: FB_BA_SubBPrio				:= (sSubject:='BO_Obj');
			BO_Obj						: FB_BA_BO_Raw := (
											iParent						:= B,
											iProfile					:= MyProfiles.BO_Prf,
											bEnPublish					:= TRUE
										); 
	{endregion}
	{region 'Multistate'}
		M								: FB_BA_View := (
											iParent						:= THIS^,
											sDescription				:= '{Multistate objects}'
										);
			 
			MV_Sub						: FB_BA_SubMPrio				:= (sSubject:='MV_Obj');
			MV_Obj						: FB_BA_MV := (
											iParent						:= M,
											iProfile					:= MyProfiles.MV_Prf,
											bEnPublish					:= TRUE
										);
			MVOp_Sub					: FB_BA_SubMV_Op				:= (sSubject:='MVOp_Obj');
			MVOp_Obj					: FB_BA_MV_Op := (
											iParent						:= M,
											iProfile					:= MyProfiles.MVOp_Prf,
											bEnPublish					:= TRUE,
											nValueRm					:= 2
										);
			MI_Sub						: FB_BA_SubMI					:= (sSubject:='MI_Obj');
			MI_Obj						: FB_BA_MI_Raw := (
											iParent						:= M,
											iProfile					:= MyProfiles.MI_Prf,
											bEnPublish					:= TRUE
										);
			MO_Sub						: FB_BA_SubMPrio				:= (sSubject:='MO_Obj');
			MO_Obj						: FB_BA_MO_Raw := (
											iParent						:= M,
											iProfile					:= MyProfiles.MO_Prf,
											bEnPublish					:= TRUE
										); 
	{endregion}
	{region 'Miscellaneous'}
		Misc							: FB_BA_View := (
											iParent						:= THIS^,
											sDescription				:= '{Miscellaneous objects}'
										);
			 
			Loop_Sub					: FB_BA_SubLoop					:= (sSubject:='Loop_Obj');
			Loop_Obj					: FB_BA_LoopSeq := (
											iParent						:= Misc,
											iProfile					:= MyProfiles.Loop_Prf,
											bEnPublish					:= TRUE,
											fProportionalConstant		:= 5.0,
											fIntegralConstant			:= 180,
											bEn							:= TRUE,
											fSetpoint					:= 20,
											fCtrlVal					:= 25
										);
	                                    
			Cal_Sub						: FB_BA_SubCal					:= (sSubject:='Cal_Obj');
			Cal_Obj						: FB_BA_Cal := (
											iParent						:= Misc,
											iProfile					:= MyProfiles.Cal_Prf,
											bEnPublish					:= TRUE,
											aDateList := [(
												eType					:= E_BA_DateValChoice.eWeekNDay,
												uDate					:= F_BA_WeekNDayVal(E_BA_Weekday.eFriday, E_BA_Week.eWeek1, E_BA_Month.eFebruary)
											)]);
												 
			SchedA_Sub					: FB_BA_SubSchedA				:= (sSubject:='SchedA_Obj');
			SchedA_Obj					: FB_BA_SchedA := (
											iParent						:= Misc,
											iProfile					:= MyProfiles.SchedA_Prf,
											bEnPublish					:= TRUE,
											aWeek						:= F_BA_SchedWeekly3xA(E_BA_Weekday.eMonday, E_BA_Weekday.eFriday, T#0H, 0.0, T#6H, 5.0, T#20H, 0.0));
			SchedB_Sub					: FB_BA_SubSchedB				:= (sSubject:='SchedB_Obj');
			SchedB_Obj					: FB_BA_SchedB := (
											iParent						:= Misc,
											iProfile					:= MyProfiles.SchedB_Prf,
											bEnPublish					:= TRUE,
											aWeek						:= F_BA_SchedWeekly3xB(E_BA_Weekday.eMonday, E_BA_Weekday.eFriday, T#0H, FALSE, T#6H, TRUE, T#20H, FALSE));
			SchedM_Sub					: FB_BA_SubSchedM				:= (sSubject:='SchedM_Obj');
			SchedM_Obj					: FB_BA_SchedM := (
											iParent						:= Misc,
											iProfile					:= MyProfiles.SchedM_Prf,
											bEnPublish					:= TRUE,
											aWeek						:= F_BA_SchedWeekly3xM(E_BA_Weekday.eMonday, E_BA_Weekday.eFriday, T#0H, 1, T#6H, 2, T#20H, 1));
												 
			Trend_Sub					: FB_BA_SubTrend				:= (sSubject:='Trend_Obj');
			Trend_Obj					: FB_BA_Trend := (
											iParent						:= Misc,
											iProfile					:= MyProfiles.Trend_Prf,
											bEnPublish					:= TRUE,
											nEventClassID				:= 11,
											stReferencedParam				:= F_BA_Reference(AV_Obj, E_BA_Parameter.ePresentValue)
										);
	{endregion}
	{region 'Custom'}
		{region 'Typed'}
			MyWthSt						: FB_BA_MyWeatherStation		:= (bEnPublish:= TRUE); 
			MyWthSt_Sub					: FB_BA_MyWeatherStationSub		:= (sSubject:='MyWthSt');
		{endregion}
		{region 'Raw'}
			MyRawWthStData				: ST_BA_MyWeatherData;
			MyRawWthSt					: FB_BA_RawPublisher;
					  
			MyRawWthStData_Sub			: ST_BA_MyWeatherData;
			MyRawWthSt_Sub				: FB_BA_RawSubscriber			:= (sSubject:='MyRawWthSt');
		{endregion}
	{endregion}
	{region 'Tests'}
		Tests							: FB_BA_View := (
											iParent						:= THIS^,
											sDescription				:= '{Test objects}'
										);
			 
		{region 'Subject path'}
			Nested1a					: FB_NestedView := (
											View						:= (iParent := Tests),
											Value						:= (bEnPublish := TRUE)
										);
			Nested1b					: FB_NestedView := (
											View						:= (iParent := Tests),
											Value						:= (bEnPublish := TRUE)
										);

			Nested1a_AV_Sub				: FB_BA_SubAV_Op := (
										//	sSubject					:= 'Value'							// -> Would lead to ambiguous subject!
											sSubject					:= 'Nested1a.Value'
										);
		{endregion}
	{endregion}
END_VAR

SUPER^(); // FB_BA_View
A(); // FB_BA_View
AO_Obj(); // FB_BA_AO_Raw
AV_Obj(); // FB_BA_AV
AI_Obj(); // FB_BA_AI_Raw
AVOp_Obj(); // FB_BA_AV_Op
AO_Sub(); // FB_BA_SubAPrio
AV_Sub(); // FB_BA_SubAPrio
AVOp_Sub(); // FB_BA_SubAV_Op
AI_Sub(); // FB_BA_SubAI
B(); // FB_BA_View
BO_Obj(); // FB_BA_BO_Raw
BV_Obj(); // FB_BA_BV
BI_Obj(); // FB_BA_BI_Raw
BVOp_Obj(); // FB_BA_BV_Op
BO_Sub(); // FB_BA_SubBPrio
BV_Sub(); // FB_BA_SubBPrio
BVOp_Sub(); // FB_BA_SubBV_Op
BI_Sub(); // FB_BA_SubBI
M(); // FB_BA_View
MO_Obj(); // FB_BA_MO_Raw
MV_Obj(); // FB_BA_MV
MI_Obj(); // FB_BA_MI_Raw
MVOp_Obj(); // FB_BA_MV_Op
MO_Sub(); // FB_BA_SubMPrio
MV_Sub(); // FB_BA_SubMPrio
MVOp_Sub(); // FB_BA_SubMV_Op
MI_Sub(); // FB_BA_SubMI
Misc(); // FB_BA_View
Loop_Obj(); // FB_BA_LoopSeq
Trend_Obj(); // FB_BA_Trend
SchedA_Obj(); // FB_BA_SchedA
SchedB_Obj(); // FB_BA_SchedB
SchedM_Obj(); // FB_BA_SchedM
Cal_Obj(); // FB_BA_Cal
Loop_Sub(); // FB_BA_SubLoop
Cal_Sub(); // FB_BA_SubCal
SchedA_Sub(); // FB_BA_SubSchedA
SchedB_Sub(); // FB_BA_SubSchedB
SchedM_Sub(); // FB_BA_SubSchedM
Trend_Sub(); // FB_BA_SubTrend
MyWthSt(); // FB_BA_MyWeatherStation
// Copy some weather data to get nice (=simulated) values - just for this demo.
MyRawWthStData := MyWthSt.stData;
MyRawWthSt(xData := MyRawWthStData); // FB_BA_RawPublisher
MyRawWthSt_Sub(xData := MyRawWthStData_Sub); // FB_BA_RawSubscriber
MyWthSt_Sub(); // FB_BA_MyWeatherStationSub
Tests(); // FB_BA_View
Nested1a(); // FB_NestedView
Nested1a_AV_Sub(); // FB_BA_SubAV_Op
Nested1b(); // FB_NestedView

END_FUNCTION_BLOCK

// ---- SAMPLES/Demo/Reference/Publish and Subscribe/FB_Ref_PubSub_Remote.TcPOU
// Example of "device-to-device" communication.
// [Notes]
// > Apply devices routes via "Diangnose / Device communication" in TerminalExplorer when PLC's are in run-mode.
//   Afterwards all communication errors will disappear. 
FUNCTION_BLOCK FB_Ref_PubSub_Remote EXTENDS FB_BA_View
VAR CONSTANT
	{region 'Test Settings'}
		// Use one (remote) device:
//		sDevice1_NetID			: T_BA_MedString				:= '192.168.10.100.1.1';
//		sDevice2_NetID			: T_BA_MedString				:= '192.168.10.100.1.1';
			 
		// Use one (loopback) device:
		sDevice1_NetID			: T_BA_MedString				:= '127.0.0.1.1.1';
		sDevice2_NetID			: T_BA_MedString				:= '127.0.0.1.1.1';
			 
		// Use two (remote and loopback) devices:
//		sDevice1_NetID			: T_BA_MedString				:= '192.168.2.200.1.1';
//		sDevice2_NetID			: T_BA_MedString				:= '127.0.0.1.1.1';
			 
		// Use two (remote) devices:
//		sDevice1_NetID			: T_BA_MedString				:= '192.168.10.100.1.1';
//		sDevice2_NetID			: T_BA_MedString				:= '192.168.2.200.1.1';
	{endregion}
END_VAR
VAR
	{region 'Analog'}
		AV_Sub					: FB_BA_SubAPrio := (
									sSubject					:= 'AV_Obj',
									sTarget						:= sDevice1_NetID,
									tReadInterval				:= T#5S								// Set shorter read interval
								);
		AVOp_Sub				: FB_BA_SubAV_Op := (
									sSubject					:= 'AVOp_Obj',
									sTarget						:= sDevice1_NetID,
									tReadInterval				:= T#5S								// Set shorter read interval
								);
		AI_Sub					: FB_BA_SubAI := (
									sSubject					:= 'AI_Obj',
									sTarget						:= sDevice2_NetID,
									tReadInterval				:= T#5S								// Set shorter read interval
								);
		AO_Sub					: FB_BA_SubAPrio := (
									sSubject					:= 'AO_Obj',
									sTarget						:= sDevice2_NetID,
									tReadInterval				:= T#5S								// Set shorter read interval
								);
	{endregion}
	{region 'Binary'}
		BV_Sub					: FB_BA_SubBPrio := (
									sSubject					:= 'BV_Obj',
									sTarget						:= sDevice1_NetID
								);
		BVOp_Sub				: FB_BA_SubBV_Op := (
									sSubject					:= 'BVOp_Obj',
									sTarget						:= sDevice1_NetID
								);
		BI_Sub					: FB_BA_SubBI := (
									sSubject					:= 'BI_Obj',
									sTarget						:= sDevice2_NetID
								);
		BO_Sub					: FB_BA_SubBPrio := (
									sSubject					:= 'BO_Obj',
									sTarget						:= sDevice2_NetID
								);
	{endregion}
	{region 'Multistate'}
		MV_Sub					: FB_BA_SubMPrio := (
									sSubject					:= 'MV_Obj',
									sTarget						:= sDevice1_NetID
								);
		MVOp_Sub				: FB_BA_SubMV_Op := (
									sSubject					:= 'MVOp_Obj',
									sTarget						:= sDevice1_NetID
								);
		MI_Sub					: FB_BA_SubMI := (
									sSubject					:= 'MI_Obj',
									sTarget						:= sDevice2_NetID
								);
		MO_Sub					: FB_BA_SubMPrio := (
									sSubject					:= 'MO_Obj',
									sTarget						:= sDevice2_NetID
								);
	{endregion}
	{region 'Multistate'}
		Loop_Sub				: FB_BA_SubLoop := (
									sSubject					:= 'Loop_Obj',
									sTarget						:= sDevice1_NetID
								);		
		Cal_Sub					: FB_BA_SubCal := (
									sSubject					:= 'Cal_Obj',
									sTarget						:= sDevice1_NetID
								);
		SchedA_Sub				: FB_BA_SubSchedA := (
									sSubject					:= 'SchedA_Obj',
									sTarget						:= sDevice1_NetID
								);
		SchedB_Sub				: FB_BA_SubSchedB := (
									sSubject					:= 'SchedB_Obj',
									sTarget						:= sDevice1_NetID
								);
		SchedM_Sub				: FB_BA_SubSchedM := (
									sSubject					:= 'SchedM_Obj',
									sTarget						:= sDevice1_NetID
								);
		Trend_Sub				: FB_BA_SubTrend := (
									sSubject					:= 'Trend_Obj',
									sTarget						:= sDevice2_NetID
								);
	{endregion}	  
	{region 'Custom'}
		{region 'Typed'}  
			MyWthSt1_Sub		: FB_BA_MyWeatherStationSub := (
									sSubject					:= 'MyWthSt',
									sTarget						:= sDevice1_NetID,
									tReadInterval				:= T#5S,							// Set shorter read interval
									tReadTolerance				:= T#20S,							// Tolerate read errors for a short time
									bClearOnReadError			:= TRUE								// Clear data on error
								);
			MyWthSt2_Sub		: FB_BA_MyWeatherStationSub := (
									sSubject					:= 'MyWthSt',
									sTarget						:= sDevice2_NetID
								);
			MyWthSt3_Sub		: FB_BA_MyWeatherStationSub := (
									sSubject					:= 'MyWthSt',
									sTarget						:= sDevice2_NetID
								);
		{endregion}
		{region 'Raw'}
			MyRawWthSt1Data_Sub	: ST_BA_MyWeatherData;
			MyRawWthSt1_Sub		: FB_BA_RawSubscriber := (
									sSubject					:= 'MyRawWthSt',
									sTarget						:= sDevice1_NetID
								);
			MyRawWthSt2Data_Sub	: ST_BA_MyWeatherData;
			MyRawWthSt2_Sub		: FB_BA_RawSubscriber := (
									sSubject					:= 'MyRawWthSt',
									sTarget						:= sDevice2_NetID
								);
		{endregion}
	{endregion} 
	{region 'Tests'}
		{region 'Subject path'}
			Nested1a_AV_Sub		: FB_BA_SubAV_Op := (
								//	sSubject					:= 'fbAV',							// -> Would lead to ambiguous subject!
									sSubject					:= 'Nested1a.Value',
									sTarget						:= sDevice1_NetID
								);
			Nested1b_AV_Sub		: FB_BA_SubAV_Op := (
								//	sSubject					:= 'fbAV',							// -> Would lead to ambiguous subject!
									sSubject					:= 'Nested1b.Value',
									sTarget						:= sDevice1_NetID
								);
		{endregion}
	{endregion}
END_VAR

SUPER^(); // FB_BA_View
AO_Sub(); // FB_BA_SubAPrio
AV_Sub(); // FB_BA_SubAPrio
AVOp_Sub(); // FB_BA_SubAV_Op
AI_Sub(); // FB_BA_SubAI
MyWthSt3_Sub(); // FB_BA_MyWeatherStationSub
BO_Sub(); // FB_BA_SubBPrio
BV_Sub(); // FB_BA_SubBPrio
BVOp_Sub(); // FB_BA_SubBV_Op
BI_Sub(); // FB_BA_SubBI
MO_Sub(); // FB_BA_SubMPrio
MV_Sub(); // FB_BA_SubMPrio
MVOp_Sub(); // FB_BA_SubMV_Op
MI_Sub(); // FB_BA_SubMI
Loop_Sub(); // FB_BA_SubLoop
Cal_Sub(); // FB_BA_SubCal
SchedA_Sub(); // FB_BA_SubSchedA
SchedB_Sub(); // FB_BA_SubSchedB
SchedM_Sub(); // FB_BA_SubSchedM
Trend_Sub(); // FB_BA_SubTrend
Nested1a_AV_Sub(); // FB_BA_SubAV_Op
MyRawWthSt1_Sub(xData := MyRawWthSt1Data_Sub); // FB_BA_RawSubscriber
MyWthSt1_Sub(); // FB_BA_MyWeatherStationSub
Nested1b_AV_Sub(); // FB_BA_SubAV_Op
MyWthSt2_Sub(); // FB_BA_MyWeatherStationSub
MyRawWthSt2_Sub(xData := MyRawWthSt2Data_Sub); // FB_BA_RawSubscriber

END_FUNCTION_BLOCK

// ---- SAMPLES/Demo/Event/FB_Evt_EventClasses.TcPOU
FUNCTION_BLOCK FB_Evt_EventClasses EXTENDS FB_BA_View
VAR
	{region 'Standard'}
		// Intention:				Demonstration of a standard use-case:
		//							- Declaration of event classes for desired event-types and alarm-modes.
		//							  (See "FB_BA_EC01" for complete example of this standard use-case).
		//							- Applies event behaviour that just works.
		EC_Std01					: FB_BA_EC := (
										iParent							:= THIS^,
										nInstanceID						:= 200,
										sDescription					:= '{Standard EC (Extended Alarm)}',
										eEventType						:= E_BA_EventType.eAlarm,
										eAlarmMode						:= E_BA_AlarmMode.eExtended
									);
		EC_Std02					: FB_BA_EC := (
										iParent							:= THIS^,
										nInstanceID						:= 201,
										sDescription					:= '{Standard EC (Standard Alarm)}',
										eEventType						:= E_BA_EventType.eAlarm,
										eAlarmMode						:= E_BA_AlarmMode.eStandard
									);
		EC_Std03					: FB_BA_EC := (
										iParent							:= THIS^,
										nInstanceID						:= 202,
										sDescription					:= '{Standard EC (Simple Alarm)}',
										eEventType						:= E_BA_EventType.eAlarm,
										eAlarmMode						:= E_BA_AlarmMode.eSimple
									);

		// Intention:				Assignment of an object's event class reference.
		SimpleAlm01					: FB_BA_BI := (
										iParent							:= THIS^,
										sDescription					:= '{Some simple alarm}',
										nEventClassID					:= 202,
										sInactiveText					:= 'Normal',
										sActiveText						:= 'Alarm'
									);
	{endregion}
	{region 'Customize default settings'}
		// Intention:				Demonstration of customizing events default behaviour by settings modification:
		//							- No difference in code to "standard use-case".
		//							  (Use implementation of the same event classes)
		//							- The following parameters are editable per alarm-mode (See "BA_Param"):
		//							  - Acknowledge Flags
		//							  - Event Enable Flags
		
		// Sample:					How to adjust the default-settings of event-classes?
		//							- No acknowledgement should be required for any "simple" events.
		//							  BA_Param.aAckFlags_Simple := [ FALSE, FALSE, FALSE ];
	{endregion}
	{region 'Individual parameters'}
		// Intention:				Demonstration of customizing individual event-classes and objects:
		// 							- Initialization of an event-classes "AcknowledgeRequired" flags.
		EC_Cstm01					: FB_BA_EC := (
										iParent							:= THIS^,
										nInstanceID						:= 220,
										sDescription					:= '{Customized EC (Alarm 1)}',
										eEventType						:= E_BA_EventType.eAlarm,
										eAlarmMode						:= E_BA_AlarmMode.UserDefined,
										aAcknowledgeRequired			:= [ TRUE, TRUE, TRUE ]
									);
		EC_Cstm02					: FB_BA_EC := (
										iParent							:= THIS^,
										nInstanceID						:= 221,
										sDescription					:= '{Customized EC (Alarm 2)}',
										eEventType						:= E_BA_EventType.eAlarm,
										eAlarmMode						:= E_BA_AlarmMode.UserDefined,
										aAcknowledgeRequired			:= [ TRUE, FALSE, FALSE ]
									);
		EC_Cstm03					: FB_BA_EC := (
										iParent							:= THIS^,
										nInstanceID						:= 222,
										sDescription					:= '{Customized EC (Alarm 3)}',
										eEventType						:= E_BA_EventType.eAlarm,
										eAlarmMode						:= E_BA_AlarmMode.UserDefined,
										aAcknowledgeRequired			:= [ FALSE, FALSE, FALSE ]
									);
										 
		// Sample:					How to initialize individual objects?
		// Intention:				- Assignment of an object's event class reference.
		// 							- Initialization of an object's "EventEnable" flags.
		Alm01						: FB_BA_BI := (
										iParent							:= THIS^,
										sDescription					:= '{Some alarm without acknowledgement}',
										nEventClassID					:= 222,
										aEventEnable					:= [ TRUE, TRUE, FALSE ],
										sInactiveText					:= 'Normal',
										sActiveText						:= 'Alarm'
									);
		Alm02						: FB_BA_BI := (
										iParent							:= THIS^,
										sDescription					:= '{Some alarm with acknowledgement}',
										nEventClassID					:= 220,
										aEventEnable					:= [ TRUE, TRUE, TRUE ],
										sInactiveText					:= 'Normal',
										sActiveText						:= 'Alarm'
									);
	{endregion}
END_VAR

EC_Cstm03(); // FB_BA_EC
EC_Std02(); // FB_BA_EC
EC_Std03(); // FB_BA_EC
EC_Cstm02(); // FB_BA_EC
SimpleAlm01(); // FB_BA_BI
EC_Cstm01(); // FB_BA_EC
Alm01(); // FB_BA_BI
Alm02(); // FB_BA_BI
SUPER^(); // FB_BA_View
EC_Std01(); // FB_BA_EC

END_FUNCTION_BLOCK

// ---- SAMPLES/Demo/Event/FB_Evt_Events.TcPOU
// Examples of objects that refer different event classes.
// > One object per 'EventType' and 'AlarmMode'.
// > One "PlantLock" per 'EventType'.
// > One "PlantLock" for entire view.
// > See "FB_BA_EC01" to view decleared event classes.
// [Hint]
// > All reference-variables are implemented to ease monitoring of relevant variables.
FUNCTION_BLOCK FB_Evt_Events EXTENDS FB_BA_View
VAR
	{region 'General'}
		Lock					: FB_BA_PlantLock				:= (iParent:=THIS^);
	{endregion}
		 
	{region 'Alarm'}
		Alm						: FB_BA_View					:= (iParent:=THIS^,	sDescription:='{Alarm}');
			AlmLock				: FB_BA_PlantLock				:= (iParent:=Alm);
							
			BIAlmSmpl_Val		: REFERENCE TO BOOL				REF= BIAlmSmpl.bVal;
			BIAlmSmpl_LockPrio	: POINTER TO E_BA_LockPriority	:= ADR(BIAlmSmpl.eEnPlantLock);
			BIAlmSmpl			: FB_BA_BI						:= (iParent:=Alm,	iLabel:=MyLabels.Cmd,	iProfile:=MyProfiles.CmdB,	nEventClassID:=12);
			BIAlmStd_Val		: REFERENCE TO BOOL				REF= BIAlmStd.bVal;
			BIAlmStd_LockPrio	: POINTER TO E_BA_LockPriority	:= ADR(BIAlmStd.eEnPlantLock);
			BIAlmStd			: FB_BA_BI						:= (iParent:=Alm,	iLabel:=MyLabels.Cmd,	iProfile:=MyProfiles.CmdB,	nEventClassID:=11,	eEnPlantLock:= E_BA_LockPriority.eHigh);
			BIAlmExt_Val		: REFERENCE TO BOOL				REF= BIAlmExt.bVal;
			BIAlmExt_LockPrio	: POINTER TO E_BA_LockPriority	:= ADR(BIAlmExt.eEnPlantLock);
			BIAlmExt			: FB_BA_BI						:= (iParent:=Alm,	iLabel:=MyLabels.Cmd,	iProfile:=MyProfiles.CmdB,	nEventClassID:=10);
	{endregion}
	{region 'Disturb'}
		Dstb					: FB_BA_View					:= (iParent:=THIS^,	sDescription:='{Disturb}');
			DstbLock			: FB_BA_PlantLock				:= (iParent:=Dstb);

			BIDstbSmpl_Val		: REFERENCE TO BOOL				REF= BIDstbSmpl.bVal;
			BIDstbSmpl_LockPrio	: POINTER TO E_BA_LockPriority	:= ADR(BIDstbSmpl.eEnPlantLock);
			BIDstbSmpl			: FB_BA_BI						:= (iParent:=Dstb,	iLabel:=MyLabels.Cmd,	iProfile:=MyProfiles.CmdB,	nEventClassID:=52);
			BIDstbStd_Val		: REFERENCE TO BOOL				REF= BIDstbStd.bVal;
			BIDstbStd_LockPrio	: POINTER TO E_BA_LockPriority	:= ADR(BIDstbStd.eEnPlantLock);
			BIDstbStd			: FB_BA_BI						:= (iParent:=Dstb,	iLabel:=MyLabels.Cmd,	iProfile:=MyProfiles.CmdB,	nEventClassID:=51,	eEnPlantLock:= E_BA_LockPriority.eMedium);
			BIDstbExt_Val		: REFERENCE TO BOOL				REF= BIDstbExt.bVal;
			BIDstbExt_LockPrio	: POINTER TO E_BA_LockPriority	:= ADR(BIDstbExt.eEnPlantLock);
			BIDstbExt			: FB_BA_BI						:= (iParent:=Dstb,	iLabel:=MyLabels.Cmd,	iProfile:=MyProfiles.CmdB,	nEventClassID:=50);
	{endregion}
	{region 'Maintenance'}
		Mntn					: FB_BA_View					:= (iParent:=THIS^,	sDescription:='{Maintenance}');
			MntnLock			: FB_BA_PlantLock				:= (iParent:=Mntn);

			BIMntnSmpl_Val		: REFERENCE TO BOOL				REF= BIMntnSmpl.bVal;
			BIMntnSmpl_LockPrio	: POINTER TO E_BA_LockPriority	:= ADR(BIMntnSmpl.eEnPlantLock);
			BIMntnSmpl			: FB_BA_BI						:= (iParent:=Mntn,	iLabel:=MyLabels.Cmd,	iProfile:=MyProfiles.CmdB,	nEventClassID:=92);
			BIMntnStd_Val		: REFERENCE TO BOOL				REF= BIMntnStd.bVal;
			BIMntnStd_LockPrio	: POINTER TO E_BA_LockPriority	:= ADR(BIMntnStd.eEnPlantLock);
			BIMntnStd			: FB_BA_BI						:= (iParent:=Mntn,	iLabel:=MyLabels.Cmd,	iProfile:=MyProfiles.CmdB,	nEventClassID:=91,	eEnPlantLock:= E_BA_LockPriority.eLocalHigh);
			BIMntnExt_Val		: REFERENCE TO BOOL				REF= BIMntnExt.bVal;
			BIMntnExt_LockPrio	: POINTER TO E_BA_LockPriority	:= ADR(BIMntnExt.eEnPlantLock);
			BIMntnExt			: FB_BA_BI						:= (iParent:=Mntn,	iLabel:=MyLabels.Cmd,	iProfile:=MyProfiles.CmdB,	nEventClassID:=90);
	{endregion}
	{region 'Notification'}
		Ntfy					: FB_BA_View					:= (iParent:=THIS^,	sDescription:='{Notification}');
			NtfyLock			: FB_BA_PlantLock				:= (iParent:=Ntfy);

			BINtfySmpl_Val		: REFERENCE TO BOOL				REF= BINtfySmpl.bVal;
			BINtfySmpl_LockPrio	: POINTER TO E_BA_LockPriority	:= ADR(BINtfySmpl.eEnPlantLock);
			BINtfySmpl			: FB_BA_BI						:= (iParent:=Ntfy,	iLabel:=MyLabels.Cmd,	iProfile:=MyProfiles.CmdB,	nEventClassID:=132);
			BINtfyStd_Val		: REFERENCE TO BOOL				REF= BINtfyStd.bVal;
			BINtfyStd_LockPrio	: POINTER TO E_BA_LockPriority	:= ADR(BINtfyStd.eEnPlantLock);
			BINtfyStd			: FB_BA_BI						:= (iParent:=Ntfy,	iLabel:=MyLabels.Cmd,	iProfile:=MyProfiles.CmdB,	nEventClassID:=131,	eEnPlantLock:= E_BA_LockPriority.eLocalMedium);
	{endregion}
	{region 'Other'}
		Other					: FB_BA_View					:= (iParent:=THIS^,	sDescription:='{Other}');
			OtherLock			: FB_BA_PlantLock				:= (iParent:=Other);
				 
			BIOthrSmpl_Val		: REFERENCE TO BOOL				REF= BIOthrSmpl.bVal;
			BIOthrSmpl_LockPrio	: POINTER TO E_BA_LockPriority	:= ADR(BIOthrSmpl.eEnPlantLock);
			BIOthrSmpl			: FB_BA_BI						:= (iParent:=Other,	iLabel:=MyLabels.Cmd,	iProfile:=MyProfiles.CmdB,	nEventClassID:=182);
			BIOthrStd_Val		: REFERENCE TO BOOL				REF= BIOthrStd.bVal;
			BIOthrStd_LockPrio	: POINTER TO E_BA_LockPriority	:= ADR(BIOthrStd.eEnPlantLock);
			BIOthrStd			: FB_BA_BI						:= (iParent:=Other,	iLabel:=MyLabels.Cmd,	iProfile:=MyProfiles.CmdB,	nEventClassID:=181);
	{endregion}                                                
END_VAR

SUPER^(); // FB_BA_View
Lock(); // FB_BA_PlantLock
Alm(); // FB_BA_View
AlmLock(); // FB_BA_PlantLock
BIAlmSmpl(); // FB_BA_BI
BIAlmStd(); // FB_BA_BI
BIAlmExt(); // FB_BA_BI
Dstb(); // FB_BA_View
DstbLock(); // FB_BA_PlantLock
BIDstbSmpl(); // FB_BA_BI
BIDstbStd(); // FB_BA_BI
BIDstbExt(); // FB_BA_BI
Mntn(); // FB_BA_View
MntnLock(); // FB_BA_PlantLock
BIMntnSmpl(); // FB_BA_BI
BIMntnStd(); // FB_BA_BI
BIMntnExt(); // FB_BA_BI
Ntfy(); // FB_BA_View
NtfyLock(); // FB_BA_PlantLock
BINtfySmpl(); // FB_BA_BI
BINtfyStd(); // FB_BA_BI
Other(); // FB_BA_View
OtherLock(); // FB_BA_PlantLock
BIOthrSmpl(); // FB_BA_BI
BIOthrStd(); // FB_BA_BI

END_FUNCTION_BLOCK

// ---- SAMPLES/Demo/Event/FB_Evt_Ack.TcPOU
// Acknowledgement-Examples.
// > One object per demonstrated 'AlarmMode'.
// > See "FB_BA_EC01" to view decleared event classes.
// [Hint]
// > All reference-variables are implemented to ease monitoring of relevant variables.
FUNCTION_BLOCK FB_Evt_Ack EXTENDS FB_BA_View
VAR               
	{region 'General'}
		bAlm_Test						: BOOL;																						// Trigger alarm for testing.
		bAlm_AckAll						: REFERENCE TO BOOL							REF= THIS^.bAcknowledgeRm;						// Acknowledge all test objects.
		bAlm_AckMode					: POINTER TO BOOL							:= ADR(BA_Param.eEvtMgmt_AckMode);				// Used reset mode (See parameter description for more details)
	{endregion}
		 
	{region 'Simple'}
		// Intention:					Alarm that automatically disappears.
		// State on active alarm:		- "bEvent = TRUE'
		//								- "stAckedTransitions = [FALSE,true,true]'
		// State when disappeared:		- "bEvent = false'
		//								- "stAckedTransitions = [true,true,true]'
		AlmSimple_Ack					: REFERENCE TO BOOL							REF= AlmSimple.bAcknowledgeRm;
		AlmSimple_Indicated				: BOOL;
		AlmSimple_Event					: REFERENCE TO BOOL							REF= AlmSimple.bEvent;
		AlmSimple						: FB_BA_BI_Raw := (
											iParent									:= THIS^,
											sInactiveText							:= 'Normal',
											sActiveText								:= 'Alarm',
											nEventClassID							:= 12);
	{endregion}
	{region 'Standard'}
		// Intention:					Alarm that is just indicated (by acknowledge transition) when disappeared.
		// State on active alarm:		- "bEvent = TRUE'
		//								- "stAckedTransitions = [FALSE,true,true]'
		// State when disappeared:		- "bEvent = false'
		//								- "stAckedTransitions = [FALSE,true,true]'
		// State after acknowledgement:	- "bEvent = false'
		//								- "stAckedTransitions = [true,true,true]'
		AlmStandard_Ack					: REFERENCE TO BOOL							REF= AlmStandard.bAcknowledgeRm;
		AlmStandard_Indicated			: BOOL;
		AlmStandard_Event				: REFERENCE TO BOOL							REF= AlmStandard.bEvent;
		AlmStandard						: FB_BA_BI_Raw := (
											iParent									:= THIS^,
											sInactiveText							:= 'Normal',
											sActiveText								:= 'Alarm',
											nEventClassID							:= 11);	
	{endregion}
	{region 'Extended'}
		// Intention:					Alarm that is indicated (by acknowledge transition) and hold when disappeared.
		//								The 'bEvent' is released when an additional reset has been triggered.
		// State on active alarm:		- "bEvent = TRUE'
		//								- "stAckedTransitions = [FALSE,true,FALSE]'
		// State when disappeared:		- "bEvent = TRUE'
		//								- "stAckedTransitions = [FALSE,true,FALSE]'
		// State after acknowledgement:	- "bEvent = TRUE'
		//								- "stAckedTransitions = [true,true,FALSE]'
		// State after reset:			- "bEvent = false'
		//								- "stAckedTransitions = [true,true,true]'
		AlmExtended_Ack					: REFERENCE TO BOOL							REF= AlmExtended.bAcknowledgeRm;
		AlmExtended_Indicated			: BOOL;
		AlmExtended_Event				: REFERENCE TO BOOL							REF= AlmExtended.bEvent;
		AlmExtended						: FB_BA_BI_Raw := (
											iParent									:= THIS^,
											sInactiveText							:= 'Normal',
											sActiveText								:= 'Alarm',
											nEventClassID							:= 10);	
	{endregion}	
END_VAR

SUPER^();

AlmSimple(bRawVal:=bAlm_Test);
AlmSimple_Indicated := (NOT AlmSimple.stAckedTransitions.bToOffnormal);
AlmStandard(bRawVal:=bAlm_Test);
AlmStandard_Indicated := (NOT AlmStandard.stAckedTransitions.bToOffnormal);
AlmExtended(bRawVal:=bAlm_Test);
AlmExtended_Indicated := (NOT AlmExtended.stAckedTransitions.bToOffnormal);

END_FUNCTION_BLOCK

// ---- SAMPLES/Demo/Event/FB_Evt_Misc.TcPOU
FUNCTION_BLOCK FB_Evt_Misc EXTENDS FB_BA_View
VAR
	{region 'Iteration'}
		// Intention:			Iterate over active events.
		bIterate				: BOOL;
		bIterate_ShowTimestamp	: BOOL				:= FALSE;
		bIterate_ShowType		: BOOL				:= TRUE;
		bIterate_ShowState		: BOOL				:= TRUE;
	{endregion}
END_VAR
VAR
	_i						: DINT;
	_sVal					: T_MaxString;
	_iObj					: I_BA_EventObject;
	_fbMsg					: FB_BA_DecorString;
END_VAR

IF (bIterate) THEN
	bIterate := FALSE;
	
	_i := F_BA_GetEventCount();
	IF (_i = 0) THEN
		F_BA_LogMessage(ADSLOG_MSGTYPE_HINT, 'EM06', 'No active events found yet.');
	ELSE
		F_BA_LogMessage1(ADSLOG_MSGTYPE_HINT, 'EM08', 'Active events: %d', F_DINT(_i));
		
		// Iterate over all active events:
		_i := 0;
		_iObj := 0;								// [Hint] Temporary iterator-object must be NULL to start iteration from the beginning.
		WHILE (F_BA_IterateEvents(_iObj)) DO
			_i := (_i+1);
			
			// Format message:
			_fbMsg.Reset();
			IF (bIterate_ShowTimestamp) THEN
				_sVal := TO_STRING(F_BA_ToDT(_iObj.EventChangeTime));
				_fbMsg.AddDecor1('%s', F_STRING(_sVal));
			END_IF
			IF (bIterate_ShowType) THEN
				_fbMsg.AddDecor1('Type: %s', F_STRINGEx(BA_EnumEN.aEventType[_iObj.EventIcon.eEventType].sName));
			END_IF
			IF (bIterate_ShowState) THEN
				_fbMsg.AddDecor1('State: %s', F_STRINGEx(BA_EnumEN.aEventIconState[_iObj.EventIcon.eState].sDescription));
			END_IF
			_fbMsg.Finish();
			
			_sVal := _iObj.ObjectName;
			F_BA_LogMessage3(ADSLOG_MSGTYPE_HINT, 'EM32', '%d. %s   %s', F_DINT(_i), F_STRING(_sVal), F_STRING(_fbMsg.sOutput));
		END_WHILE
	END_IF
END_IF

END_FUNCTION_BLOCK

// ---- SAMPLES/Demo/Structure/FB_Struct_Nested.TcPOU
// Examples of nested objects and possible variants for initialization of parent/child-relations.
FUNCTION_BLOCK FB_Struct_Nested EXTENDS FB_BA_View
VAR
	{region 'Variant 1'}
		Nested1a		: FB_NestedView				:= (View:=(iParent:=THIS^));
		Nested1b		: FB_NestedView				:= (View:=(iParent:=THIS^));
	{endregion}
	{region 'Variant 2'}
		Nested2			: FB_NestedView2			(THIS^);     
	{endregion}
END_VAR

SUPER^();

// Variant 1:
Nested1a();
Nested1b();

// Variant 2:
Nested2();

END_FUNCTION_BLOCK

// ---- SAMPLES/Demo/[Helper]/FunctionBlocks/Nested/FB_NestedView2.TcPOU
FUNCTION_BLOCK FB_NestedView2
VAR_INPUT CONSTANT
	Enable	: FB_BA_BV_Op := (
				iProfile		:= MyProfiles.BVOp_Prf,
				bValueRm		:= FALSE
			);		
	Value	: FB_BA_AV_Op := (
				iProfile		:= MyProfiles.AVOp_Prf,
				fValueRm		:= 0.0
			);	
END_VAR

Enable();
Value();

METHOD FB_init : BOOL
VAR_INPUT
	bInitRetains : BOOL; // if TRUE, the retain variables are initialized (warm start / cold start)
	bInCopyCode : BOOL;  // if TRUE, the instance afterwards gets moved into the copy code (online change)
END_VAR
VAR_INPUT
	iParent : I_BA_View;
END_VAR
Enable.Parent := iParent;
Value.Parent := iParent;
END_METHOD

END_FUNCTION_BLOCK

// ---- SAMPLES/Demo/Plant/FB_Plt_Init1.TcPOU
// How to initialize plant control at declaration (Recommended workflow).
// [Hint]
// > All reference-variables are implemented to ease monitoring of relevant variables.
FUNCTION_BLOCK FB_Plt_Init1 EXTENDS FB_BA_View
VAR
   	{region 'Aggregates'}
		DmprSu_Open							: REFERENCE TO BOOL							REF= DmprSu.bOpen;
		DmprSu_Val							: REFERENCE TO REAL							REF= DmprSu.fActiveVal;
		DmprSu								: FB_TimerAggregateA						:= (iParent:=THIS^,					iLabel:=MyLabels.DmprSu);
		FanSu_Val							: REFERENCE TO UDINT						REF= FanSu.nActiveVal;
		FanSu								: FB_BA_AggregateM							:= (iParent:=THIS^,					iLabel:=MyLabels.FanSu);
			 
		DmprEx_Open							: REFERENCE TO BOOL							REF= DmprEx.bOpen;
		DmprEx_Val							: REFERENCE TO REAL							REF= DmprEx.fActiveVal;
		DmprEx								: FB_TimerAggregateA						:= (iParent:=THIS^,					iLabel:=MyLabels.DmprEx);
		FanEx_Val							: REFERENCE TO UDINT						REF= FanEx.nActiveVal;
		FanEx								: FB_BA_AggregateM							:= (iParent:=THIS^,					iLabel:=MyLabels.FanEx);
			 
